KUKA KRL program: MyProgram_258().src

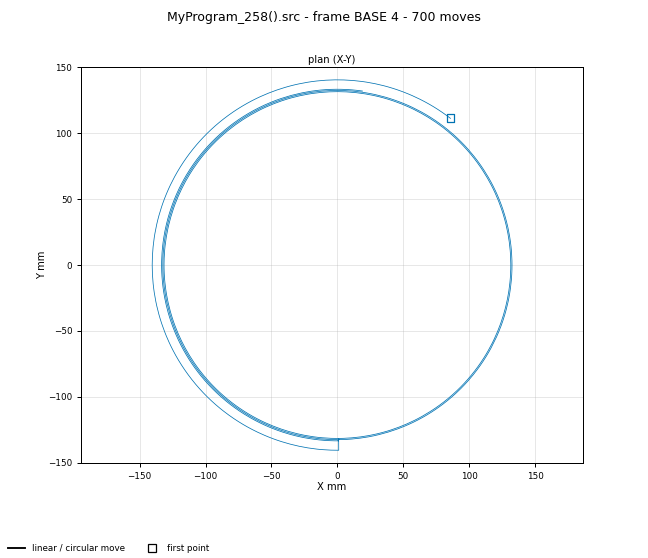
[picture p0: tool path of MyProgram_258().src in frame BASE 4, 700 of 700 moves have a stored position in this frame; points joined in program order, loops and branches not executed]
&ACCESS RVP
&REL 1
&PARAM TEMPLATE = C:\KRC\Roboter\Template\vorgabe
&PARAM EDITMASK = *
DEF MyProgram_258()
; ---- Setting reference (Base) ----
$BASE = BASE_DATA[4]

; --------------------------
; ---- Setting tool (TCP) ----
$TOOL = TOOL_DATA[3]
; --------------------------

$VEL.CP = VEL_APROX_PRINT
Startdeposition()
$VEL.CP = VEL_PRINT
LIN {X 85.7174,Y 111.2402,Z 166,A 52.9681,B 10.7255,C 0.0747,E1 10.8235,E2 398.079} C_DIS
LIN {X 83.0634,Y 113.235,Z 166,A 54.4984,B 10.7255,C 0.0678,E1 10.82,E2 396.526} C_DIS
LIN {X 79.5534,Y 115.7279,Z 166,A 56.2475,B 10.7255,C 0.0651,E1 10.816,E2 394.7774} C_DIS
LIN {X 75.9568,Y 118.12,Z 166,A 57.9765,B 10.7255,C 0.0632,E1 10.812,E2 393.0524} C_DIS
LIN {X 72.9306,Y 120.0121,Z 166,A 59.3925,B 10.7255,C 0.0621,E1 10.8086,E2 391.6413} C_DIS
LIN {X 69.966,Y 121.7647,Z 166,A 60.8768,B 10.7255,C 0.0581,E1 10.805,E2 390.1468} C_DIS
LIN {X 66.2006,Y 123.8518,Z 166,A 62.5606,B 10.7255,C 0.0575,E1 10.8009,E2 388.4721} C_DIS
LIN {X 62.4847,Y 125.7655,Z 166,A 64.2605,B 10.7256,C 0.0555,E1 10.7967,E2 386.7727} C_DIS
LIN {X 59.1907,Y 127.3486,Z 166,A 65.6969,B 10.7256,C 0.055,E1 10.7931,E2 385.3432} C_DIS
LIN {X 56.6753,Y 128.4896,Z 166,A 66.832,B 10.7256,C 0.0535,E1 10.7902,E2 384.2072} C_DIS
LIN {X 53.7331,Y 129.7462,Z 166,A 68.1368,B 10.7256,C 0.0521,E1 10.7868,E2 382.9025} C_DIS
LIN {X 49.8023,Y 131.3058,Z 166,A 69.9999,B 10.7256,C 0.0469,E1 10.7819,E2 381.0219} C_DIS
LIN {X 45.6873,Y 132.7929,Z 166,A 71.6306,B 10.7256,C 0.0491,E1 10.7777,E2 379.4111} C_DIS
LIN {X 42.4057,Y 133.877,Z 166,A 73.0559,B 10.7256,C 0.0475,E1 10.7739,E2 377.9841} C_DIS
LIN {X 38.7409,Y 134.9848,Z 166,A 74.5834,B 10.7256,C 0.0472,E1 10.7698,E2 376.4612} C_DIS
LIN {X 35.4064,Y 135.8978,Z 166,A 76.0506,B 10.7256,C 0.0448,E1 10.7658,E2 374.9871} C_DIS
LIN {X 31.4821,Y 136.8581,Z 166,A 77.4069,B 10.7256,C 0.0508,E1 10.7622,E2 373.6681} C_DIS
LIN {X 28.7539,Y 137.4591,Z 166,A 78.7425,B 10.7256,C 0.0454,E1 10.7585,E2 372.308} C_DIS
LIN {X 25.6831,Y 138.0655,Z 166,A 80.0395,B 10.7256,C 0.0443,E1 10.755,E2 371.0088} C_DIS
LIN {X 22.2954,Y 138.6535,Z 166,A 81.461,B 10.7256,C 0.0432,E1 10.751,E2 369.5854} C_DIS
LIN {X 18.6465,Y 139.1895,Z 166,A 82.9581,B 10.7256,C 0.0429,E1 10.7469,E2 368.0897} C_DIS
LIN {X 14.9704,Y 139.6322,Z 166,A 84.3565,B 10.7256,C 0.0451,E1 10.7431,E2 366.7061} C_DIS
LIN {X 11.786,Y 139.937,Z 166,A 85.7616,B 10.7256,C 0.0424,E1 10.7391,E2 365.2888} C_DIS
LIN {X 8.3535,Y 140.1841,Z 166,A 87.1286,B 10.7256,C 0.0431,E1 10.7353,E2 363.927} C_DIS
LIN {X 4.9167,Y 140.3475,Z 166,A 88.5506,B 10.7256,C 0.0426,E1 10.7314,E2 362.5033} C_DIS
LIN {X 1.7237,Y 140.4233,Z 166,A 89.9324,B 10.7256,C 0.0407,E1 10.7275,E2 361.1121} C_DIS
LIN {X -1.7428,Y 140.423,Z 166,A 91.3065,B 10.7256,C 0.0418,E1 10.7237,E2 359.7437} C_DIS
LIN {X -5.4304,Y 140.3274,Z 166,A 92.7483,B 10.7256,C 0.0434,E1 10.7197,E2 358.3106} C_DIS
LIN {X -8.7826,Y 140.1576,Z 166,A 94.1374,B 10.7256,C 0.0433,E1 10.7158,E2 356.9198} C_DIS
LIN {X -12.3639,Y 139.8881,Z 166,A 95.6189,B 10.7256,C 0.0433,E1 10.7116,E2 355.437} C_DIS
LIN {X -15.5753,Y 139.5671,Z 166,A 96.9396,B 10.7256,C 0.0437,E1 10.708,E2 354.1166} C_DIS
LIN {X -19.209,Y 139.1139,Z 166,A 98.4595,B 10.7256,C 0.0437,E1 10.7038,E2 352.5943} C_DIS
LIN {X -22.5934,Y 138.6039,Z 166,A 99.8716,B 10.7256,C 0.0441,E1 10.6999,E2 351.1811} C_DIS
LIN {X -26.0391,Y 137.9974,Z 166,A 101.2635,B 10.7256,C 0.0457,E1 10.6961,E2 349.7946} C_DIS
LIN {X -29.3329,Y 137.3349,Z 166,A 102.6588,B 10.7256,C 0.046,E1 10.6922,E2 348.397} C_DIS
LIN {X -32.6927,Y 136.5739,Z 166,A 104.0676,B 10.7256,C 0.0469,E1 10.6884,E2 346.9887} C_DIS
LIN {X -36.0321,Y 135.731,Z 166,A 105.4187,B 10.7256,C 0.0493,E1 10.6848,E2 345.6455} C_DIS
LIN {X -39.5794,Y 134.7392,Z 166,A 106.9465,B 10.7256,C 0.05,E1 10.6807,E2 344.1156} C_DIS
LIN {X -42.9868,Y 133.6913,Z 166,A 108.3925,B 10.7256,C 0.0515,E1 10.6768,E2 342.6718} C_DIS
LIN {X -45.9258,Y 132.7102,Z 166,A 109.7162,B 10.7256,C 0.0514,E1 10.6733,E2 341.3415} C_DIS
LIN {X -49.682,Y 131.3509,Z 166,A 111.2836,B 10.7256,C 0.0545,E1 10.6692,E2 339.7834} C_DIS
LIN {X -52.371,Y 130.3013,Z 166,A 112.5376,B 10.7256,C 0.0541,E1 10.6659,E2 338.5205} C_DIS
LIN {X -55.8214,Y 128.8608,Z 166,A 113.9843,B 10.7256,C 0.0577,E1 10.6623,E2 337.0851} C_DIS
LIN {X -58.4834,Y 127.6757,Z 166,A 115.2991,B 10.7256,C 0.0564,E1 10.6589,E2 335.7554} C_DIS
LIN {X -61.664,Y 126.1703,Z 166,A 116.7076,B 10.7256,C 0.0589,E1 10.6553,E2 334.3516} C_DIS
LIN {X -64.8452,Y 124.5651,Z 166,A 118.1373,B 10.7256,C 0.0614,E1 10.6518,E2 332.9262} C_DIS
LIN {X -68.498,Y 122.5963,Z 166,A 119.9049,B 10.7256,C 0.0623,E1 10.6474,E2 331.1507} C_DIS
LIN {X -72.1926,Y 120.4576,Z 166,A 121.6574,B 10.7256,C 0.0647,E1 10.6432,E2 329.3985} C_DIS
LIN {X -75.871,Y 118.1749,Z 166,A 123.4185,B 10.7256,C 0.0676,E1 10.6391,E2 327.6397} C_DIS
LIN {X -78.8459,Y 116.2112,Z 166,A 125.0176,B 10.7256,C 0.0669,E1 10.6353,E2 326.0236} C_DIS
LIN {X -82.7583,Y 113.4589,Z 166,A 126.9317,B 10.7256,C 0.0711,E1 10.631,E2 324.1162} C_DIS
LIN {X -86.3102,Y 110.7807,Z 166,A 128.7237,B 10.7255,C 0.0749,E1 10.627,E2 322.3288} C_DIS
LIN {X -89.1917,Y 108.4744,Z 166,A 130.3265,B 10.7255,C 0.0757,E1 10.6235,E2 320.7152} C_DIS
LIN {X -92.4731,Y 105.6904,Z 166,A 132.0844,B 10.7255,C 0.0791,E1 10.6198,E2 318.9588} C_DIS
LIN {X -95.6725,Y 102.803,Z 166,A 133.7492,B 10.7255,C 0.0846,E1 10.6164,E2 317.3077} C_DIS
LIN {X -98.6977,Y 99.903,Z 166,A 135.4739,B 10.7254,C 0.0879,E1 10.613,E2 315.5829} C_DIS
LIN {X -101.6253,Y 96.9226,Z 166,A 137.2193,B 10.7254,C 0.0907,E1 10.6096,E2 313.8341} C_DIS
LIN {X -104.1361,Y 94.2199,Z 166,A 138.7083,B 10.7254,C 0.0943,E1 10.6068,E2 312.3488} C_DIS
LIN {X -106.8373,Y 91.1457,Z 166,A 140.4303,B 10.7254,C 0.097,E1 10.6036,E2 310.6219} C_DIS
LIN {X -109.1132,Y 88.4087,Z 166,A 142.0079,B 10.7254,C 0.0976,E1 10.6008,E2 309.03} C_DIS
LIN {X -112.0478,Y 84.6581,Z 166,A 143.9057,B 10.7253,C 0.1032,E1 10.5976,E2 307.14} C_DIS
LIN {X -114.3919,Y 81.4632,Z 166,A 145.5929,B 10.7253,C 0.1056,E1 10.5948,E2 305.4456} C_DIS
LIN {X -116.8357,Y 77.9173,Z 166,A 147.3595,B 10.7252,C 0.1097,E1 10.592,E2 303.6797} C_DIS
LIN {X -119.1097,Y 74.3951,Z 166,A 149.0835,B 10.7252,C 0.1137,E1 10.5895,E2 301.9559} C_DIS
LIN {X -121.334,Y 70.71,Z 166,A 150.7899,B 10.7251,C 0.1193,E1 10.587,E2 300.2578} C_DIS
LIN {X -123.4441,Y 66.9578,Z 166,A 152.6788,B 10.7251,C 0.121,E1 10.5845,E2 298.354} C_DIS
LIN {X -125.2195,Y 63.5706,Z 166,A 154.115,B 10.725,C 0.1277,E1 10.5827,E2 296.9353} C_DIS
LIN {X -126.6897,Y 60.5875,Z 166,A 155.2897,B 10.725,C 0.1351,E1 10.5813,E2 295.7852} C_DIS
LIN {X -128.075,Y 57.6021,Z 166,A 156.8232,B 10.725,C 0.1348,E1 10.5795,E2 294.229} C_DIS
LIN {X -129.665,Y 53.9275,Z 166,A 158.5396,B 10.7249,C 0.1375,E1 10.5776,E2 292.5039} C_DIS
LIN {X -131.0262,Y 50.5316,Z 166,A 160.0242,B 10.7249,C 0.1418,E1 10.576,E2 291.022} C_DIS
LIN {X -132.2233,Y 47.3105,Z 166,A 161.4457,B 10.7248,C 0.1453,E1 10.5747,E2 289.5996} C_DIS
LIN {X -133.3465,Y 44.0455,Z 166,A 162.8717,B 10.7248,C 0.1489,E1 10.5734,E2 288.173} C_DIS
LIN {X -134.4583,Y 40.5278,Z 166,A 164.4487,B 10.7247,C 0.1516,E1 10.5721,E2 286.5885} C_DIS
LIN {X -135.3443,Y 37.4599,Z 166,A 165.7163,B 10.7247,C 0.1561,E1 10.5712,E2 285.3268} C_DIS
LIN {X -136.2255,Y 34.1176,Z 166,A 167.1446,B 10.7246,C 0.1597,E1 10.5702,E2 283.8977} C_DIS
LIN {X -137.0215,Y 30.7667,Z 166,A 168.5675,B 10.7246,C 0.1634,E1 10.5693,E2 282.4742} C_DIS
LIN {X -137.7352,Y 27.397,Z 166,A 169.9898,B 10.7245,C 0.1671,E1 10.5685,E2 281.0512} C_DIS
LIN {X -138.3664,Y 24.0105,Z 166,A 171.4122,B 10.7245,C 0.1708,E1 10.5678,E2 279.6282} C_DIS
LIN {X -138.9138,Y 20.6098,Z 166,A 172.9305,B 10.7244,C 0.1726,E1 10.5671,E2 278.097} C_DIS
LIN {X -139.407,Y 16.9421,Z 166,A 174.34,B 10.7243,C 0.1791,E1 10.5666,E2 276.7019} C_DIS
LIN {X -139.7635,Y 13.6928,Z 166,A 175.7816,B 10.7243,C 0.1807,E1 10.5662,E2 275.2479} C_DIS
LIN {X -140.0738,Y 10.0321,Z 166,A 177.2439,B 10.7242,C 0.1859,E1 10.5659,E2 273.7919} C_DIS
LIN {X -140.2655,Y 6.8493,Z 166,A 178.5857,B 10.7242,C 0.1888,E1 10.5657,E2 272.4462} C_DIS
LIN {X -140.4085,Y 2.6106,Z 166,A -179.8067,B 10.724,C 0.1965,E1 10.5656,E2 270.8561} C_DIS
LIN {X -140.4365,Y -0.0242,Z 166,A -178.4973,B 10.724,C 0.1948,E1 10.5656,E2 269.5179} C_DIS
LIN {X -140.3907,Y -3.4567,Z 166,A -177.1039,B 10.724,C 0.199,E1 10.5656,E2 268.1267} C_DIS
LIN {X -140.266,Y -6.8381,Z 166,A -175.7478,B 10.7238,C 0.2035,E1 10.5658,E2 266.7751} C_DIS
LIN {X -139.9886,Y -11.1743,Z 166,A -174.043,B 10.7238,C 0.2101,E1 10.5661,E2 265.0808} C_DIS
LIN {X -139.7327,Y -14.0133,Z 166,A -172.8116,B 10.7237,C 0.2121,E1 10.5665,E2 263.8418} C_DIS
LIN {X -139.3773,Y -17.1908,Z 166,A -171.436,B 10.7237,C 0.2144,E1 10.5669,E2 262.4583} C_DIS
LIN {X -138.8773,Y -20.8502,Z 166,A -169.9239,B 10.7235,C 0.2186,E1 10.5675,E2 260.947} C_DIS
LIN {X -138.2783,Y -24.503,Z 166,A -168.4632,B 10.7235,C 0.224,E1 10.5682,E2 259.494} C_DIS
LIN {X -137.685,Y -27.6437,Z 166,A -167.077,B 10.7234,C 0.226,E1 10.5689,E2 258.0985} C_DIS
LIN {X -136.9287,Y -31.1727,Z 166,A -165.623,B 10.7234,C 0.2306,E1 10.5698,E2 256.6481} C_DIS
LIN {X -136.0361,Y -34.8636,Z 166,A -164.0961,B 10.7232,C 0.2354,E1 10.5708,E2 255.1255} C_DIS
LIN {X -135.342,Y -37.4682,Z 166,A -162.9018,B 10.7232,C 0.2365,E1 10.5717,E2 253.9199} C_DIS
LIN {X -134.3111,Y -41.0087,Z 166,A -161.3782,B 10.7231,C 0.2403,E1 10.5729,E2 252.3951} C_DIS
LIN {X -133.2661,Y -44.2868,Z 166,A -159.9559,B 10.7231,C 0.2438,E1 10.5742,E2 250.9716} C_DIS
LIN {X -132.1411,Y -47.5382,Z 166,A -158.534,B 10.7229,C 0.2472,E1 10.5755,E2 249.5485} C_DIS
LIN {X -130.9367,Y -50.7616,Z 166,A -157.0359,B 10.7229,C 0.249,E1 10.577,E2 248.0393} C_DIS
LIN {X -129.6473,Y -53.9697,Z 166,A -155.5789,B 10.7229,C 0.2518,E1 10.5786,E2 246.5775} C_DIS
LIN {X -127.7265,Y -58.3735,Z 166,A -153.6315,B 10.7227,C 0.2573,E1 10.5808,E2 244.6333} C_DIS
LIN {X -126.2024,Y -61.599,Z 166,A -152.2299,B 10.7226,C 0.2622,E1 10.5825,E2 243.2396} C_DIS
LIN {X -124.5972,Y -64.7841,Z 166,A -150.7803,B 10.7225,C 0.2661,E1 10.5843,E2 241.7917} C_DIS
LIN {X -122.6149,Y -68.4648,Z 166,A -148.9967,B 10.7225,C 0.2687,E1 10.5867,E2 239.9993} C_DIS
LIN {X -120.4574,Y -72.1929,Z 166,A -147.1417,B 10.7224,C 0.2709,E1 10.5893,E2 238.1328} C_DIS
LIN {X -118.111,Y -75.9708,Z 166,A -145.269,B 10.7223,C 0.2741,E1 10.5922,E2 236.2537} C_DIS
LIN {X -115.7286,Y -79.5524,Z 166,A -143.5007,B 10.7222,C 0.2779,E1 10.5949,E2 234.4846} C_DIS
LIN {X -113.2061,Y -83.1027,Z 166,A -141.7158,B 10.7221,C 0.2819,E1 10.5978,E2 232.6996} C_DIS
LIN {X -110.479,Y -86.6953,Z 166,A -139.881,B 10.722,C 0.2861,E1 10.601,E2 230.8665} C_DIS
LIN {X -107.5054,Y -90.3564,Z 166,A -137.994,B 10.7218,C 0.2912,E1 10.6043,E2 228.9854} C_DIS
LIN {X -104.6071,Y -93.6965,Z 166,A -136.1896,B 10.7218,C 0.295,E1 10.6076,E2 227.1817} C_DIS
LIN {X -101.7035,Y -96.8408,Z 166,A -134.3395,B 10.7218,C 0.2963,E1 10.6112,E2 225.3188} C_DIS
LIN {X -98.6888,Y -99.9119,Z 166,A -132.5285,B 10.7216,C 0.2986,E1 10.6148,E2 223.5014} C_DIS
LIN {X -95.5786,Y -102.8905,Z 166,A -130.851,B 10.7216,C 0.3037,E1 10.6182,E2 221.8349} C_DIS
LIN {X -92.3556,Y -105.7928,Z 166,A -129.0546,B 10.7214,C 0.3064,E1 10.6219,E2 220.0355} C_DIS
LIN {X -89.088,Y -108.5591,Z 166,A -127.3599,B 10.7214,C 0.3107,E1 10.6256,E2 218.3481} C_DIS
LIN {X -86.3015,Y -110.7874,Z 166,A -125.75,B 10.7214,C 0.3097,E1 10.6291,E2 216.7185} C_DIS
LIN {X -82.3699,Y -113.7404,Z 166,A -123.764,B 10.7212,C 0.3135,E1 10.6336,E2 214.7356} C_DIS
LIN {X -78.5505,Y -116.4111,Z 166,A -121.8547,B 10.7212,C 0.3163,E1 10.638,E2 212.8257} C_DIS
LIN {X -75.1269,Y -118.6494,Z 166,A -120.1443,B 10.7211,C 0.3178,E1 10.642,E2 211.11} C_DIS
LIN {X -71.4556,Y -120.8964,Z 166,A -118.5045,B 10.7209,C 0.3229,E1 10.6459,E2 209.4857} C_DIS
LIN {X -68.3612,Y -122.6727,Z 166,A -116.8962,B 10.7209,C 0.3214,E1 10.6499,E2 207.8575} C_DIS
LIN {X -64.569,Y -124.7101,Z 166,A -115.1164,B 10.7209,C 0.323,E1 10.6543,E2 206.0747} C_DIS
LIN {X -60.6866,Y -126.6424,Z 166,A -113.492,B 10.7208,C 0.3284,E1 10.6583,E2 204.4693} C_DIS
LIN {X -57.686,Y -128.0375,Z 166,A -112.3048,B 10.7206,C 0.3337,E1 10.6613,E2 203.3034} C_DIS
LIN {X -55.323,Y -129.0763,Z 166,A -111.0698,B 10.7207,C 0.3306,E1 10.6645,E2 202.0446} C_DIS
LIN {X -52.1431,Y -130.3932,Z 166,A -109.6601,B 10.7207,C 0.3319,E1 10.6681,E2 200.6342} C_DIS
LIN {X -48.9322,Y -131.6317,Z 166,A -108.249,B 10.7207,C 0.333,E1 10.6718,E2 199.222} C_DIS
LIN {X -45.6787,Y -132.7958,Z 166,A -106.8356,B 10.7207,C 0.3341,E1 10.6756,E2 197.8079} C_DIS
LIN {X -42.3173,Y -133.9052,Z 166,A -105.3701,B 10.7206,C 0.3347,E1 10.6795,E2 196.3394} C_DIS
LIN {X -38.8146,Y -134.9632,Z 166,A -103.9003,B 10.7206,C 0.3363,E1 10.6834,E2 194.8725} C_DIS
LIN {X -35.7228,Y -135.8135,Z 166,A -102.5809,B 10.7206,C 0.3369,E1 10.687,E2 193.5514} C_DIS
LIN {X -31.9412,Y -136.7532,Z 166,A -101.0442,B 10.7205,C 0.3391,E1 10.6911,E2 192.0213} C_DIS
LIN {X -29.0661,Y -137.3925,Z 166,A -99.784,B 10.7205,C 0.3383,E1 10.6946,E2 190.7531} C_DIS
LIN {X -25.6925,Y -138.0637,Z 166,A -98.3811,B 10.7205,C 0.3389,E1 10.6984,E2 189.3499} C_DIS
LIN {X -22.3036,Y -138.6522,Z 166,A -96.9553,B 10.7205,C 0.3389,E1 10.7024,E2 187.9208} C_DIS
LIN {X -18.6541,Y -139.1885,Z 166,A -95.4474,B 10.7205,C 0.3392,E1 10.7065,E2 186.412} C_DIS
LIN {X -15.465,Y -139.5789,Z 166,A -94.1374,B 10.7205,C 0.3395,E1 10.7102,E2 185.1016} C_DIS
LIN {X -11.7927,Y -139.9364,Z 166,A -92.6422,B 10.7205,C 0.3399,E1 10.7143,E2 183.6071} C_DIS
LIN {X -8.3593,Y -140.1837,Z 166,A -91.2738,B 10.7204,C 0.3409,E1 10.7181,E2 182.2429} C_DIS
LIN {X -4.9207,Y -140.3473,Z 166,A -89.8498,B 10.7204,C 0.3404,E1 10.7221,E2 180.8157} C_DIS
LIN {X -1.71,Y -140.4235,Z 166,A -88.4652,B 10.7204,C 0.3385,E1 10.726,E2 179.4207} C_DIS
LIN {X 0.9985,Y -140.4282,Z 166,A -87.7382,B 10.7202,C 0.3476,E1 10.7279,E2 178.7427} C_DIS
Enddeposition()
LIN {X 0.9528,Y -131.4631,Z 167,A -88.3932,B 11.3356,C 0.2691,E1 11.3404,E2 178.9455} C_DIS
Startdeposition()
$VEL.CP = VEL_PRINT
LIN {X -1.6196,Y -131.4601,Z 167,A -89.776,B 11.3354,C 0.2755,E1 11.3364,E2 180.3603} C_DIS
LIN {X -4.8405,Y -131.38,Z 167,A -91.1508,B 11.3354,C 0.2748,E1 11.3326,E2 181.7322} C_DIS
LIN {X -8.4656,Y -131.1965,Z 167,A -92.6004,B 11.3355,C 0.2717,E1 11.3286,E2 183.1667} C_DIS
LIN {X -11.6768,Y -130.9506,Z 167,A -94.0267,B 11.3355,C 0.2721,E1 11.3246,E2 184.5963} C_DIS
LIN {X -14.4963,Y -130.6678,Z 167,A -95.3539,B 11.3355,C 0.274,E1 11.3209,E2 185.935} C_DIS
LIN {X -18.0814,Y -130.2204,Z 167,A -96.8808,B 11.3355,C 0.2725,E1 11.3167,E2 187.4567} C_DIS
LIN {X -21.2806,Y -129.7354,Z 167,A -98.2888,B 11.3355,C 0.272,E1 11.3128,E2 188.8648} C_DIS
LIN {X -24.4682,Y -129.1718,Z 167,A -99.5735,B 11.3355,C 0.2685,E1 11.3093,E2 190.1348} C_DIS
LIN {X -27.6142,Y -128.5358,Z 167,A -101.1,B 11.3355,C 0.2708,E1 11.3051,E2 191.677} C_DIS
LIN {X -30.3791,Y -127.9112,Z 167,A -102.3409,B 11.3355,C 0.2702,E1 11.3017,E2 192.9189} C_DIS
LIN {X -33.8824,Y -127.0274,Z 167,A -103.9798,B 11.3355,C 0.2707,E1 11.2972,E2 194.5657} C_DIS
LIN {X -37.0063,Y -126.1527,Z 167,A -105.3341,B 11.3355,C 0.2684,E1 11.2936,E2 195.9132} C_DIS
LIN {X -39.7094,Y -125.3284,Z 167,A -106.5704,B 11.3356,C 0.2676,E1 11.2903,E2 197.1502} C_DIS
LIN {X -42.7754,Y -124.3153,Z 167,A -107.9828,B 11.3356,C 0.2666,E1 11.2866,E2 198.5634} C_DIS
LIN {X -45.8088,Y -123.2299,Z 167,A -109.392,B 11.3356,C 0.2654,E1 11.2829,E2 199.9733} C_DIS
LIN {X -48.8167,Y -122.0696,Z 167,A -110.802,B 11.3356,C 0.2642,E1 11.2792,E2 201.384} C_DIS
LIN {X -51.8039,Y -120.8323,Z 167,A -112.2163,B 11.3357,C 0.2629,E1 11.2756,E2 202.799} C_DIS
LIN {X -54.7506,Y -119.5262,Z 167,A -113.6279,B 11.3357,C 0.2615,E1 11.272,E2 204.2114} C_DIS
LIN {X -57.8494,Y -118.0571,Z 167,A -115.0803,B 11.3358,C 0.2588,E1 11.2683,E2 205.6587} C_DIS
LIN {X -60.8996,Y -116.5127,Z 167,A -116.4678,B 11.3359,C 0.2548,E1 11.2649,E2 207.0339} C_DIS
LIN {X -64.05,Y -114.8138,Z 167,A -118.31,B 11.3359,C 0.259,E1 11.2603,E2 208.9097} C_DIS
LIN {X -67.5842,Y -112.7693,Z 167,A -119.9987,B 11.3359,C 0.2545,E1 11.2563,E2 210.5874} C_DIS
LIN {X -70.671,Y -110.8608,Z 167,A -121.6957,B 11.3359,C 0.2547,E1 11.2522,E2 212.2979} C_DIS
LIN {X -74.39,Y -108.4,Z 167,A -123.6086,B 11.3359,C 0.2511,E1 11.2478,E2 214.2068} C_DIS
LIN {X -77.0224,Y -106.5458,Z 167,A -124.9509,B 11.3361,C 0.2475,E1 11.2448,E2 215.5415} C_DIS
LIN {X -80.0944,Y -104.2564,Z 167,A -126.6676,B 11.3361,C 0.2457,E1 11.2409,E2 217.2633} C_DIS
LIN {X -83.2482,Y -101.7555,Z 167,A -128.4689,B 11.3361,C 0.2437,E1 11.237,E2 219.0697} C_DIS
LIN {X -86.4707,Y -99.0316,Z 167,A -130.3006,B 11.3362,C 0.2402,E1 11.2331,E2 220.9} C_DIS
LIN {X -89.4839,Y -96.3177,Z 167,A -132.0835,B 11.3362,C 0.2371,E1 11.2295,E2 222.6842} C_DIS
LIN {X -92.3941,Y -93.5302,Z 167,A -133.9462,B 11.3363,C 0.2359,E1 11.2257,E2 224.5588} C_DIS
LIN {X -95.3517,Y -90.5132,Z 167,A -135.8075,B 11.3363,C 0.2326,E1 11.2221,E2 226.4216} C_DIS
LIN {X -98.3569,Y -87.2376,Z 167,A -137.6719,B 11.3365,C 0.227,E1 11.2186,E2 228.2766} C_DIS
LIN {X -101.2512,Y -83.8608,Z 167,A -139.6968,B 11.3365,C 0.2246,E1 11.215,E2 230.3107} C_DIS
LIN {X -104.0256,Y -80.3937,Z 167,A -141.5014,B 11.3367,C 0.2176,E1 11.2119,E2 232.0988} C_DIS
LIN {X -105.9668,Y -77.8169,Z 167,A -143.0743,B 11.3367,C 0.2178,E1 11.2092,E2 233.6906} C_DIS
LIN {X -108.6249,Y -74.0623,Z 167,A -144.9383,B 11.3368,C 0.2102,E1 11.2063,E2 235.537} C_DIS
LIN {X -110.294,Y -71.5519,Z 167,A -146.3582,B 11.3368,C 0.2092,E1 11.2041,E2 236.9685} C_DIS
LIN {X -112.1328,Y -68.6344,Z 167,A -147.8428,B 11.3368,C 0.2052,E1 11.2019,E2 238.45} C_DIS
LIN {X -113.7899,Y -65.8505,Z 167,A -149.2653,B 11.337,C 0.2019,E1 11.1999,E2 239.8728} C_DIS
LIN {X -115.3682,Y -63.0446,Z 167,A -150.5965,B 11.337,C 0.1969,E1 11.1981,E2 241.1945} C_DIS
LIN {X -116.8769,Y -60.2004,Z 167,A -152.146,B 11.337,C 0.1963,E1 11.196,E2 242.7602} C_DIS
LIN {X -118.1647,Y -57.6313,Z 167,A -153.4289,B 11.337,C 0.1937,E1 11.1945,E2 244.0459} C_DIS
LIN {X -119.7507,Y -54.2596,Z 167,A -154.9749,B 11.3372,C 0.1878,E1 11.1927,E2 245.5815} C_DIS
LIN {X -120.9894,Y -51.4404,Z 167,A -156.3794,B 11.3372,C 0.1856,E1 11.1911,E2 246.9923} C_DIS
LIN {X -122.2209,Y -48.4413,Z 167,A -157.8015,B 11.3372,C 0.1819,E1 11.1896,E2 248.4144} C_DIS
LIN {X -123.3708,Y -45.4326,Z 167,A -159.2278,B 11.3373,C 0.1786,E1 11.1882,E2 249.8422} C_DIS
LIN {X -124.4468,Y -42.3962,Z 167,A -160.6477,B 11.3373,C 0.1751,E1 11.1869,E2 251.2629} C_DIS
LIN {X -125.649,Y -38.6824,Z 167,A -162.5181,B 11.3374,C 0.1737,E1 11.1853,E2 253.1516} C_DIS
LIN {X -126.7149,Y -35.0351,Z 167,A -164.0453,B 11.3375,C 0.1665,E1 11.1842,E2 254.6622} C_DIS
LIN {X -127.6297,Y -31.5469,Z 167,A -165.7364,B 11.3375,C 0.1645,E1 11.183,E2 256.3659} C_DIS
LIN {X -128.3549,Y -28.4521,Z 167,A -167.0588,B 11.3376,C 0.1593,E1 11.1822,E2 257.6797} C_DIS
LIN {X -128.9411,Y -25.6615,Z 167,A -168.2945,B 11.3376,C 0.1556,E1 11.1815,E2 258.9134} C_DIS
LIN {X -129.5291,Y -22.5087,Z 167,A -169.7075,B 11.3377,C 0.1519,E1 11.1808,E2 260.3269} C_DIS
LIN {X -130.0472,Y -19.2933,Z 167,A -171.1719,B 11.3377,C 0.1487,E1 11.1801,E2 261.7952} C_DIS
LIN {X -130.5424,Y -15.5789,Z 167,A -172.7879,B 11.3378,C 0.1436,E1 11.1796,E2 263.4075} C_DIS
LIN {X -130.8365,Y -12.8823,Z 167,A -174.0944,B 11.3378,C 0.1426,E1 11.1792,E2 264.7274} C_DIS
LIN {X -131.1127,Y -9.6697,Z 167,A -175.4356,B 11.3379,C 0.1372,E1 11.1789,E2 266.0597} C_DIS
LIN {X -131.33,Y -6.063,Z 167,A -176.9873,B 11.3379,C 0.1321,E1 11.1787,E2 267.6072} C_DIS
LIN {X -131.4446,Y -2.5537,Z 167,A -178.6248,B 11.3379,C 0.1298,E1 11.1785,E2 269.2556} C_DIS
LIN {X -131.4667,Y 0.7845,Z 167,A 179.8914,B 11.338,C 0.1261,E1 11.1785,E2 270.7413} C_DIS
LIN {X -131.3681,Y 5.147,Z 167,A 178.0051,B 11.338,C 0.1202,E1 11.1787,E2 272.6237} C_DIS
LIN {X -131.1977,Y 8.4457,Z 167,A 176.6123,B 11.3382,C 0.115,E1 11.1789,E2 274.0096} C_DIS
LIN {X -130.9508,Y 11.6749,Z 167,A 175.1443,B 11.3382,C 0.112,E1 11.1793,E2 275.4827} C_DIS
LIN {X -130.6588,Y 14.5795,Z 167,A 173.7611,B 11.3382,C 0.1105,E1 11.1797,E2 276.8774} C_DIS
LIN {X -130.2126,Y 18.1359,Z 167,A 172.2485,B 11.3382,C 0.1049,E1 11.1802,E2 278.3825} C_DIS
LIN {X -129.7327,Y 21.297,Z 167,A 170.8374,B 11.3382,C 0.1012,E1 11.1808,E2 279.7941} C_DIS
LIN {X -129.1745,Y 24.4542,Z 167,A 169.5469,B 11.3383,C 0.095,E1 11.1815,E2 281.0707} C_DIS
LIN {X -128.528,Y 27.6503,Z 167,A 167.9884,B 11.3383,C 0.0936,E1 11.1824,E2 282.6436} C_DIS
LIN {X -127.909,Y 30.3884,Z 167,A 166.7412,B 11.3383,C 0.0906,E1 11.1831,E2 283.8921} C_DIS
LIN {X -127.0251,Y 33.8909,Z 167,A 165.2467,B 11.3384,C 0.0845,E1 11.1842,E2 285.3755} C_DIS
LIN {X -126.2662,Y 36.6186,Z 167,A 163.8979,B 11.3384,C 0.0832,E1 11.1852,E2 286.7364} C_DIS
LIN {X -125.3302,Y 39.7039,Z 167,A 162.4751,B 11.3384,C 0.0796,E1 11.1864,E2 288.1596} C_DIS
LIN {X -124.3192,Y 42.7642,Z 167,A 161.053,B 11.3384,C 0.076,E1 11.1877,E2 289.5822} C_DIS
LIN {X -123.2341,Y 45.7975,Z 167,A 159.629,B 11.3384,C 0.0725,E1 11.189,E2 291.0068} C_DIS
LIN {X -122.0036,Y 48.9805,Z 167,A 158.1656,B 11.3385,C 0.0679,E1 11.1905,E2 292.4658} C_DIS
LIN {X -120.8275,Y 51.8149,Z 167,A 156.7749,B 11.3385,C 0.0653,E1 11.192,E2 293.8612} C_DIS
LIN {X -119.5263,Y 54.7504,Z 167,A 155.3549,B 11.3385,C 0.0619,E1 11.1936,E2 295.282} C_DIS
LIN {X -118.1452,Y 57.6709,Z 167,A 153.9342,B 11.3385,C 0.0584,E1 11.1954,E2 296.7026} C_DIS
LIN {X -116.4688,Y 60.9832,Z 167,A 152.4919,B 11.3386,C 0.0506,E1 11.1972,E2 298.1226} C_DIS
LIN {X -115.1796,Y 63.3893,Z 167,A 151.092,B 11.3386,C 0.0517,E1 11.1991,E2 299.5456} C_DIS
LIN {X -113.5928,Y 66.1911,Z 167,A 149.6609,B 11.3386,C 0.0486,E1 11.2011,E2 300.9783} C_DIS
LIN {X -111.9361,Y 68.9551,Z 167,A 148.1718,B 11.3386,C 0.0468,E1 11.2032,E2 302.4757} C_DIS
LIN {X -109.5762,Y 72.6476,Z 167,A 146.2018,B 11.3386,C 0.0432,E1 11.2062,E2 304.4505} C_DIS
LIN {X -107.2584,Y 76.0275,Z 167,A 144.574,B 11.3386,C 0.0356,E1 11.2088,E2 306.0579} C_DIS
LIN {X -105.5966,Y 78.3189,Z 167,A 143.1404,B 11.3386,C 0.0367,E1 11.2112,E2 307.5133} C_DIS
LIN {X -103.1467,Y 81.5191,Z 167,A 141.3473,B 11.3386,C 0.0333,E1 11.2143,E2 309.3087} C_DIS
LIN {X -100.4654,Y 84.8014,Z 167,A 139.4835,B 11.3386,C 0.0294,E1 11.2176,E2 311.1724} C_DIS
LIN {X -97.8204,Y 87.8386,Z 167,A 137.7229,B 11.3386,C 0.0255,E1 11.2209,E2 312.9317} C_DIS
LIN {X -95.0841,Y 90.7935,Z 167,A 135.9585,B 11.3387,C 0.0219,E1 11.2242,E2 314.6952} C_DIS
LIN {X -91.9484,Y 93.9678,Z 167,A 134.0438,B 11.3387,C 0.0172,E1 11.228,E2 316.6045} C_DIS
LIN {X -88.8833,Y 96.8721,Z 167,A 132.1318,B 11.3387,C 0.0149,E1 11.2319,E2 318.5229} C_DIS
LIN {X -85.8738,Y 99.5497,Z 167,A 130.3725,B 11.3387,C 0.0115,E1 11.2356,E2 320.2807} C_DIS
LIN {X -82.7725,Y 102.1433,Z 167,A 128.5482,B 11.3387,C 0.0094,E1 11.2396,E2 322.1104} C_DIS
LIN {X -79.2916,Y 104.868,Z 167,A 126.7615,B 11.3387,C 0.0029,E1 11.2435,E2 323.8791} C_DIS
LIN {X -77.0136,Y 106.5522,Z 167,A 125.4468,B 11.3387,C 0.0024,E1 11.2465,E2 325.2018} C_DIS
LIN {X -74.0585,Y 108.6275,Z 167,A 123.9775,B 11.3387,C -0.0025,E1 11.2498,E2 326.6575} C_DIS
LIN {X -71.69,Y 110.2043,Z 167,A 122.6027,B 11.3387,C -0.0017,E1 11.253,E2 328.0467} C_DIS
LIN {X -68.53,Y 112.1969,Z 167,A 121.038,B 11.3387,C -0.0057,E1 11.2567,E2 329.6025} C_DIS
LIN {X -65.8044,Y 113.8166,Z 167,A 119.6477,B 11.3387,C -0.0076,E1 11.2601,E2 330.9925} C_DIS
LIN {X -62.7673,Y 115.5195,Z 167,A 118.2627,B 11.3387,C -0.0127,E1 11.2634,E2 332.3608} C_DIS
LIN {X -60.1896,Y 116.8824,Z 167,A 116.8488,B 11.3387,C -0.0114,E1 11.267,E2 333.7901} C_DIS
LIN {X -57.6673,Y 118.147,Z 167,A 115.5558,B 11.3387,C -0.0117,E1 11.2702,E2 335.0894} C_DIS
LIN {X -54.3786,Y 119.6974,Z 167,A 114.0139,B 11.3387,C -0.0147,E1 11.2741,E2 336.625} C_DIS
LIN {X -51.4313,Y 120.9934,Z 167,A 112.5912,B 11.3387,C -0.016,E1 11.2778,E2 338.0488} C_DIS
LIN {X -48.4525,Y 122.2164,Z 167,A 111.1902,B 11.3387,C -0.0176,E1 11.2814,E2 339.4484} C_DIS
LIN {X -45.4293,Y 123.372,Z 167,A 109.7663,B 11.3387,C -0.0189,E1 11.2851,E2 340.8727} C_DIS
LIN {X -42.3564,Y 124.4606,Z 167,A 108.3407,B 11.3387,C -0.0202,E1 11.2889,E2 342.2977} C_DIS
LIN {X -38.5188,Y 125.6991,Z 167,A 106.5767,B 11.3387,C -0.0217,E1 11.2936,E2 344.0612} C_DIS
LIN {X -35.0609,Y 126.7077,Z 167,A 105.0021,B 11.3387,C -0.023,E1 11.2978,E2 345.6352} C_DIS
LIN {X -31.5772,Y 127.6224,Z 167,A 103.4314,B 11.3387,C -0.0242,E1 11.302,E2 347.2049} C_DIS
LIN {X -28.8204,Y 128.2715,Z 167,A 102.1237,B 11.3387,C -0.0234,E1 11.3056,E2 348.5203} C_DIS
LIN {X -25.6459,Y 128.9442,Z 167,A 100.7757,B 11.3387,C -0.0258,E1 11.3093,E2 349.8597} C_DIS
LIN {X -22.4753,Y 129.5351,Z 167,A 99.3678,B 11.3387,C -0.0266,E1 11.3131,E2 351.2669} C_DIS
LIN {X -19.2808,Y 130.049,Z 167,A 97.9318,B 11.3387,C -0.0266,E1 11.3171,E2 352.7051} C_DIS
LIN {X -15.6987,Y 130.5281,Z 167,A 96.3658,B 11.3387,C -0.0276,E1 11.3214,E2 354.269} C_DIS
LIN {X -12.8824,Y 130.8365,Z 167,A 95.0472,B 11.3387,C -0.0261,E1 11.3251,E2 355.5966} C_DIS
LIN {X -9.2633,Y 131.1424,Z 167,A 93.608,B 11.3387,C -0.0298,E1 11.3291,E2 357.0184} C_DIS
LIN {X -6.0472,Y 131.3308,Z 167,A 92.1619,B 11.3387,C -0.0291,E1 11.3331,E2 358.4687} C_DIS
LIN {X -2.8271,Y 131.44,Z 167,A 90.7992,B 11.3387,C -0.0303,E1 11.3369,E2 359.8259} C_DIS
LIN {X 0.3912,Y 131.4687,Z 167,A 89.4405,B 11.3387,C -0.0314,E1 11.3407,E2 361.1788} C_DIS
LIN {X 3.6152,Y 131.4192,Z 167,A 88.0108,B 11.3387,C -0.0308,E1 11.3447,E2 362.6107} C_DIS
LIN {X 6.8517,Y 131.2904,Z 167,A 86.4628,B 11.3387,C -0.0276,E1 11.3491,E2 364.174} C_DIS
LIN {X 11.6749,Y 130.9508,Z 167,A 84.4421,B 11.3387,C -0.0292,E1 11.3547,E2 366.1838} C_DIS
LIN {X 14.4913,Y 130.6683,Z 167,A 83.1183,B 11.3387,C -0.0268,E1 11.3584,E2 367.5177} C_DIS
LIN {X 18.3984,Y 130.1751,Z 167,A 81.547,B 11.3387,C -0.0296,E1 11.3627,E2 369.0716} C_DIS
LIN {X 21.2776,Y 129.7359,Z 167,A 80.1914,B 11.3387,C -0.027,E1 11.3664,E2 370.4368} C_DIS
LIN {X 24.4518,Y 129.1749,Z 167,A 78.914,B 11.3387,C -0.0294,E1 11.3699,E2 371.699} C_DIS
LIN {X 27.6117,Y 128.5364,Z 167,A 77.3922,B 11.3387,C -0.0259,E1 11.3741,E2 373.2341} C_DIS
LIN {X 31.2848,Y 127.6929,Z 167,A 75.6104,B 11.3387,C -0.0215,E1 11.379,E2 375.0318} C_DIS
LIN {X 35.0741,Y 126.704,Z 167,A 74.0532,B 11.3387,C -0.0239,E1 11.3831,E2 376.5713} C_DIS
LIN {X 38.6885,Y 125.6471,Z 167,A 72.3213,B 11.3387,C -0.0204,E1 11.3878,E2 378.3135} C_DIS
LIN {X 42.772,Y 124.3165,Z 167,A 70.5547,B 11.3387,C -0.0213,E1 11.3924,E2 380.0677} C_DIS
LIN {X 45.8054,Y 123.2311,Z 167,A 69.1574,B 11.3387,C -0.0201,E1 11.3961,E2 381.4641} C_DIS
LIN {X 48.8231,Y 122.067,Z 167,A 67.7548,B 11.3387,C -0.0188,E1 11.3998,E2 382.8657} C_DIS
LIN {X 51.8012,Y 120.8335,Z 167,A 66.3581,B 11.3387,C -0.0175,E1 11.4033,E2 384.2615} C_DIS
LIN {X 54.7503,Y 119.5263,Z 167,A 64.9617,B 11.3387,C -0.0161,E1 11.4069,E2 385.6568} C_DIS
LIN {X 57.6741,Y 118.1436,Z 167,A 63.5616,B 11.3387,C -0.0146,E1 11.4104,E2 387.0558} C_DIS
LIN {X 60.8948,Y 116.5152,Z 167,A 62.1545,B 11.3387,C -0.0166,E1 11.4139,E2 388.4437} C_DIS
LIN {X 63.3906,Y 115.179,Z 167,A 60.6617,B 11.3387,C -0.0086,E1 11.4176,E2 389.9669} C_DIS
LIN {X 66.2056,Y 113.5844,Z 167,A 59.3587,B 11.3387,C -0.0092,E1 11.4207,E2 391.2576} C_DIS
LIN {X 68.9706,Y 111.9266,Z 167,A 57.8847,B 11.3387,C -0.0054,E1 11.4243,E2 392.7398} C_DIS
LIN {X 72.0442,Y 109.9734,Z 167,A 56.4564,B 11.3387,C -0.0069,E1 11.4276,E2 394.1499} C_DIS
LIN {X 74.3878,Y 108.4015,Z 167,A 55.1058,B 11.3387,C -0.0019,E1 11.4307,E2 395.5148} C_DIS
LIN {X 77.0187,Y 106.5485,Z 167,A 53.7845,B 11.3387,C -0.0016,E1 11.4337,E2 396.827} C_DIS
LIN {X 80.0882,Y 104.2611,Z 167,A 52.0951,B 11.3387,C 0.0018,E1 11.4375,E2 398.5193} C_DIS
LIN {X 83.2529,Y 101.7516,Z 167,A 50.3166,B 11.3387,C 0.0054,E1 11.4414,E2 400.3005} C_DIS
LIN {X 86.4896,Y 99.0151,Z 167,A 48.5121,B 11.3387,C 0.0078,E1 11.4452,E2 402.1006} C_DIS
LIN {X 89.4826,Y 96.3188,Z 167,A 46.7664,B 11.3387,C 0.0109,E1 11.4488,E2 403.8457} C_DIS
LIN {X 92.3923,Y 93.532,Z 167,A 44.9375,B 11.3387,C 0.0163,E1 11.4525,E2 405.6839} C_DIS
LIN {X 95.3484,Y 90.5168,Z 167,A 43.1112,B 11.3387,C 0.0198,E1 11.456,E2 407.5093} C_DIS
LIN {X 98.361,Y 87.233,Z 167,A 41.2775,B 11.3387,C 0.0212,E1 11.4594,E2 409.3312} C_DIS
LIN {X 101.01,Y 84.152,Z 167,A 39.4485,B 11.3387,C 0.0266,E1 11.4627,E2 411.1679} C_DIS
LIN {X 103.6514,Y 80.8764,Z 167,A 37.6608,B 11.3387,C 0.0295,E1 11.4658,E2 412.9512} C_DIS
LIN {X 105.8275,Y 78.0066,Z 167,A 36.0815,B 11.3387,C 0.0334,E1 11.4685,E2 414.5325} C_DIS
LIN {X 108.4111,Y 74.3738,Z 167,A 34.2763,B 11.3387,C 0.0345,E1 11.4713,E2 416.3227} C_DIS
LIN {X 110.2022,Y 71.6933,Z 167,A 32.8055,B 11.3387,C 0.0396,E1 11.4736,E2 417.802} C_DIS
LIN {X 112.1523,Y 68.6028,Z 167,A 31.3104,B 11.3387,C 0.041,E1 11.4758,E2 419.2867} C_DIS
LIN {X 113.7929,Y 65.8454,Z 167,A 29.9299,B 11.3387,C 0.0441,E1 11.4777,E2 420.666} C_DIS
LIN {X 115.3675,Y 63.046,Z 167,A 28.6315,B 11.3387,C 0.045,E1 11.4795,E2 421.9535} C_DIS
LIN {X 116.8732,Y 60.2077,Z 167,A 27.1488,B 11.3387,C 0.0507,E1 11.4814,E2 423.4468} C_DIS
LIN {X 118.1505,Y 57.66,Z 167,A 25.8675,B 11.3386,C 0.055,E1 11.483,E2 424.7337} C_DIS
LIN {X 119.6905,Y 54.3941,Z 167,A 24.3833,B 11.3386,C 0.0568,E1 11.4847,E2 426.2086} C_DIS
LIN {X 121.0003,Y 51.4152,Z 167,A 22.9743,B 11.3386,C 0.0604,E1 11.4863,E2 427.6176} C_DIS
LIN {X 122.2212,Y 48.4407,Z 167,A 21.388,B 11.3386,C 0.069,E1 11.488,E2 429.2268} C_DIS
LIN {X 123.3697,Y 45.4356,Z 167,A 20.2064,B 11.3386,C 0.0671,E1 11.4891,E2 430.3836} C_DIS
LIN {X 124.4447,Y 42.4024,Z 167,A 18.8216,B 11.3386,C 0.0705,E1 11.4904,E2 431.7675} C_DIS
LIN {X 125.6982,Y 38.5217,Z 167,A 16.9638,B 11.3385,C 0.0775,E1 11.492,E2 433.6363} C_DIS
LIN {X 126.9375,Y 34.2192,Z 167,A 15.0026,B 11.3385,C 0.0833,E1 11.4934,E2 435.6003} C_DIS
LIN {X 127.9134,Y 30.3702,Z 167,A 13.4369,B 11.3385,C 0.0839,E1 11.4945,E2 437.1481} C_DIS
LIN {X 128.7008,Y 26.842,Z 167,A 11.9407,B 11.3385,C 0.0863,E1 11.4953,E2 438.6364} C_DIS
LIN {X 129.2491,Y 24.064,Z 167,A 10.6692,B 11.3384,C 0.0908,E1 11.496,E2 439.9136} C_DIS
LIN {X 129.8013,Y 20.8859,Z 167,A 9.2093,B 11.3384,C 0.0963,E1 11.4967,E2 441.3812} C_DIS
LIN {X 130.2753,Y 17.6841,Z 167,A 7.7714,B 11.3383,C 0.1011,E1 11.4973,E2 442.8237} C_DIS
LIN {X 130.7106,Y 14.0984,Z 167,A 6.4177,B 11.3383,C 0.0999,E1 11.4977,E2 444.1528} C_DIS
LIN {X 131.0171,Y 10.8902,Z 167,A 5.0112,B 11.3383,C 0.1041,E1 11.498,E2 445.5609} C_DIS
LIN {X 131.2212,Y 8.0646,Z 167,A 3.6729,B 11.3382,C 0.1104,E1 11.4983,E2 446.9127} C_DIS
LIN {X 131.4163,Y 3.718,Z 167,A 2.0773,B 11.3382,C 0.108,E1 11.4985,E2 448.4746} C_DIS
LIN {X 131.467,Y 0.7331,Z 167,A 0.5845,B 11.3382,C 0.117,E1 11.4985,E2 449.9915} C_DIS
LIN {X 131.4399,Y -2.8368,Z 167,A -1.0783,B 11.3381,C 0.1244,E1 11.4985,E2 451.6687} C_DIS
LIN {X 131.2913,Y -6.8338,Z 167,A -2.6834,B 11.3381,C 0.1259,E1 11.4983,E2 453.2593} C_DIS
LIN {X 131.1121,Y -9.6781,Z 167,A -3.9561,B 11.338,C 0.1303,E1 11.498,E2 454.537} C_DIS
LIN {X 130.7962,Y -13.3015,Z 167,A -5.4594,B 11.338,C 0.1328,E1 11.4976,E2 456.0323} C_DIS
LIN {X 130.433,Y -16.4805,Z 167,A -6.8676,B 11.338,C 0.1373,E1 11.4972,E2 457.4436} C_DIS
LIN {X 129.9893,Y -19.6723,Z 167,A -8.249,B 11.3379,C 0.1408,E1 11.4966,E2 458.8239} C_DIS
LIN {X 129.4465,Y -22.9706,Z 167,A -9.6576,B 11.3379,C 0.1438,E1 11.496,E2 460.2282} C_DIS
LIN {X 128.895,Y -25.8877,Z 167,A -11.0059,B 11.3378,C 0.149,E1 11.4952,E2 461.5846} C_DIS
LIN {X 128.1795,Y -29.2235,Z 167,A -12.3213,B 11.3378,C 0.1487,E1 11.4944,E2 462.8811} C_DIS
LIN {X 127.4741,Y -32.1615,Z 167,A -13.763,B 11.3377,C 0.1558,E1 11.4935,E2 464.3392} C_DIS
LIN {X 126.7043,Y -35.0728,Z 167,A -15.0202,B 11.3377,C 0.1582,E1 11.4926,E2 465.5914} C_DIS
LIN {X 125.8082,Y -38.1624,Z 167,A -16.4038,B 11.3376,C 0.1617,E1 11.4915,E2 466.9743} C_DIS
LIN {X 124.8317,Y -41.2442,Z 167,A -17.7946,B 11.3376,C 0.1652,E1 11.4903,E2 468.3646} C_DIS
LIN {X 123.7836,Y -44.2907,Z 167,A -19.1802,B 11.3375,C 0.1687,E1 11.489,E2 469.7495} C_DIS
LIN {X 122.6575,Y -47.3199,Z 167,A -20.5704,B 11.3375,C 0.1721,E1 11.4876,E2 471.1392} C_DIS
LIN {X 121.4606,Y -50.313,Z 167,A -21.957,B 11.3374,C 0.1755,E1 11.4862,E2 472.5253} C_DIS
LIN {X 120.1914,Y -53.2743,Z 167,A -23.3689,B 11.3374,C 0.1796,E1 11.4846,E2 473.9397} C_DIS
LIN {X 118.8205,Y -56.2656,Z 167,A -24.7526,B 11.3373,C 0.1822,E1 11.483,E2 475.319} C_DIS
LIN {X 117.4195,Y -59.1346,Z 167,A -26.2352,B 11.3372,C 0.1883,E1 11.4811,E2 476.8141} C_DIS
LIN {X 115.6885,Y -62.4555,Z 167,A -27.7493,B 11.3372,C 0.1895,E1 11.4791,E2 478.3161} C_DIS
LIN {X 114.3876,Y -64.808,Z 167,A -28.9073,B 11.3372,C 0.1923,E1 11.4776,E2 479.4739} C_DIS
LIN {X 112.764,Y -67.5932,Z 167,A -30.3011,B 11.3371,C 0.1956,E1 11.4756,E2 480.8679} C_DIS
LIN {X 110.8628,Y -70.6679,Z 167,A -31.9729,B 11.3369,C 0.2022,E1 11.4731,E2 482.553} C_DIS
LIN {X 108.4023,Y -74.3866,Z 167,A -33.8413,B 11.3369,C 0.2051,E1 11.4702,E2 484.4147} C_DIS
LIN {X 106.5459,Y -77.0223,Z 167,A -35.1606,B 11.3369,C 0.2063,E1 11.468,E2 485.7252} C_DIS
LIN {X 104.2564,Y -80.0945,Z 167,A -36.8456,B 11.3368,C 0.2108,E1 11.4652,E2 487.414} C_DIS
LIN {X 101.7363,Y -83.2717,Z 167,A -38.6247,B 11.3368,C 0.2152,E1 11.4621,E2 489.1965} C_DIS
LIN {X 99.0142,Y -86.4906,Z 167,A -40.4174,B 11.3367,C 0.2183,E1 11.4588,E2 490.9858} C_DIS
LIN {X 96.3205,Y -89.4808,Z 167,A -42.1585,B 11.3366,C 0.222,E1 11.4556,E2 492.7273} C_DIS
LIN {X 93.512,Y -92.4124,Z 167,A -43.9962,B 11.3365,C 0.2276,E1 11.452,E2 494.5752} C_DIS
LIN {X 90.5013,Y -95.363,Z 167,A -45.8192,B 11.3365,C 0.2312,E1 11.4483,E2 496.3985} C_DIS
LIN {X 87.231,Y -98.3628,Z 167,A -47.6469,B 11.3364,C 0.2324,E1 11.4445,E2 498.2155} C_DIS
LIN {X 84.1575,Y -101.0055,Z 167,A -49.4016,B 11.3364,C 0.2357,E1 11.4408,E2 499.9706} C_DIS
LIN {X 80.8752,Y -103.6523,Z 167,A -51.2697,B 11.3362,C 0.24,E1 11.4367,E2 501.8442} C_DIS
LIN {X 77.4435,Y -106.2406,Z 167,A -53.1496,B 11.3362,C 0.2436,E1 11.4325,E2 503.7267} C_DIS
LIN {X 74.0608,Y -108.626,Z 167,A -54.8935,B 11.3362,C 0.2453,E1 11.4285,E2 505.4653} C_DIS
LIN {X 70.656,Y -110.8703,Z 167,A -56.744,B 11.336,C 0.2502,E1 11.4241,E2 507.3263} C_DIS
LIN {X 67.0014,Y -113.1167,Z 167,A -58.4078,B 11.336,C 0.2481,E1 11.4202,E2 508.9672} C_DIS
LIN {X 64.4614,Y -114.5826,Z 167,A -59.7125,B 11.336,C 0.2508,E1 11.417,E2 510.2762} C_DIS
LIN {X 61.977,Y -115.9456,Z 167,A -61.0357,B 11.336,C 0.2548,E1 11.4137,E2 511.6112} C_DIS
LIN {X 58.77,Y -117.603,Z 167,A -62.4545,B 11.336,C 0.2533,E1 11.4103,E2 513.0128} C_DIS
LIN {X 55.8285,Y -119.0278,Z 167,A -64.06,B 11.3358,C 0.2597,E1 11.4061,E2 514.6414} C_DIS
LIN {X 52.8993,Y -120.3587,Z 167,A -65.3071,B 11.3358,C 0.2577,E1 11.403,E2 515.8711} C_DIS
LIN {X 49.9382,Y -121.6171,Z 167,A -66.7114,B 11.3358,C 0.2596,E1 11.3994,E2 517.2769} C_DIS
LIN {X 47.1587,Y -122.7202,Z 167,A -68.02,B 11.3358,C 0.2612,E1 11.396,E2 518.5871} C_DIS
LIN {X 43.7624,Y -123.9732,Z 167,A -69.5475,B 11.3358,C 0.2618,E1 11.392,E2 520.1099} C_DIS
LIN {X 40.8566,Y -124.9608,Z 167,A -70.9445,B 11.3357,C 0.2647,E1 11.3883,E2 521.5152} C_DIS
LIN {X 37.907,Y -125.8863,Z 167,A -72.2889,B 11.3357,C 0.2659,E1 11.3847,E2 522.8602} C_DIS
LIN {X 33.828,Y -127.0419,Z 167,A -74.1783,B 11.3356,C 0.2686,E1 11.3796,E2 524.7559} C_DIS
LIN {X 30.0238,Y -127.9967,Z 167,A -75.7739,B 11.3356,C 0.2673,E1 11.3753,E2 526.3391} C_DIS
LIN {X 26.8393,Y -128.7014,Z 167,A -77.1401,B 11.3356,C 0.267,E1 11.3716,E2 527.6997} C_DIS
LIN {X 24.0583,Y -129.2501,Z 167,A -78.4264,B 11.3356,C 0.2691,E1 11.368,E2 528.9929} C_DIS
LIN {X 20.8821,Y -129.8019,Z 167,A -79.8726,B 11.3356,C 0.2709,E1 11.364,E2 530.445} C_DIS
LIN {X 17.6782,Y -130.2761,Z 167,A -81.3543,B 11.3355,C 0.2734,E1 11.3599,E2 531.936} C_DIS
LIN {X 14.0952,Y -130.711,Z 167,A -82.723,B 11.3355,C 0.2692,E1 11.3562,E2 533.2811} C_DIS
LIN {X 10.8856,Y -131.0175,Z 167,A -84.1457,B 11.3355,C 0.2702,E1 11.3522,E2 534.7067} C_DIS
LIN {X 8.0601,Y -131.2215,Z 167,A -85.5007,B 11.3355,C 0.2735,E1 11.3484,E2 536.0768} C_DIS
LIN {X 4.825,Y -131.3806,Z 167,A -86.9064,B 11.3355,C 0.2737,E1 11.3444,E2 537.4826} C_DIS
LIN {X 1.6022,Y -131.4604,Z 167,A -88.3625,B 11.3355,C 0.2752,E1 11.3404,E2 538.9455} C_DIS
LIN {X 1.6022,Y -131.4604,Z 167,A -88.3625,B 11.3355,C 0.2752,E1 11.3404,E2 538.9455} C_DIS
Enddeposition()
LIN {X 0.9593,Y -132.3799,Z 167,A -88.2151,B 11.3357,C 0.2719,E1 11.341,E2 538.7814} C_DIS
Startdeposition()
$VEL.CP = VEL_PRINT
LIN {X 3.625,Y -132.3348,Z 167,A -86.7635,B 11.3359,C 0.2645,E1 11.3452,E2 537.293} C_DIS
LIN {X 6.9134,Y -132.204,Z 167,A -85.2036,B 11.3359,C 0.2608,E1 11.3496,E2 535.7158} C_DIS
LIN {X 11.023,Y -131.9247,Z 167,A -83.4647,B 11.3359,C 0.2613,E1 11.3544,E2 533.9812} C_DIS
LIN {X 14.2365,Y -131.6166,Z 167,A -82.1586,B 11.3359,C 0.2629,E1 11.358,E2 532.6855} C_DIS
LIN {X 17.1893,Y -131.2636,Z 167,A -80.7974,B 11.336,C 0.2604,E1 11.3618,E2 531.3144} C_DIS
LIN {X 20.647,Y -130.7648,Z 167,A -79.3507,B 11.336,C 0.2612,E1 11.3658,E2 529.8748} C_DIS
LIN {X 23.6645,Y -130.2524,Z 167,A -78.0208,B 11.336,C 0.2602,E1 11.3695,E2 528.5434} C_DIS
LIN {X 27.53,Y -129.4907,Z 167,A -76.1652,B 11.3361,C 0.2552,E1 11.3746,E2 526.6682} C_DIS
LIN {X 31.4443,Y -128.5963,Z 167,A -74.3811,B 11.3361,C 0.2527,E1 11.3795,E2 524.8772} C_DIS
LIN {X 38.5261,Y -126.6543,Z 167,A -71.3418,B 11.3361,C 0.2532,E1 11.3876,E2 521.8526} C_DIS
LIN {X 43.4725,Y -125.0427,Z 167,A -69.4647,B 11.3361,C 0.2602,E1 11.3925,E2 520.0196} C_DIS
LIN {X 45.5125,Y -124.3163,Z 167,A -68.2653,B 11.3361,C 0.2526,E1 11.3957,E2 518.7874} C_DIS
LIN {X 48.0788,Y -123.3448,Z 167,A -67.0132,B 11.3362,C 0.2496,E1 11.399,E2 517.5263} C_DIS
LIN {X 51.1104,Y -122.1198,Z 167,A -65.6544,B 11.3362,C 0.2492,E1 11.4025,E2 516.1733} C_DIS
LIN {X 54.2767,Y -120.746,Z 167,A -64.1555,B 11.3362,C 0.2471,E1 11.4063,E2 514.6725} C_DIS
LIN {X 57.4474,Y -119.2705,Z 167,A -62.6703,B 11.3363,C 0.2458,E1 11.41,E2 513.1895} C_DIS
LIN {X 60.8054,Y -117.5963,Z 167,A -60.9162,B 11.3364,C 0.2401,E1 11.4144,E2 511.418} C_DIS
LIN {X 64.7911,Y -115.4475,Z 167,A -59.1094,B 11.3364,C 0.241,E1 11.4188,E2 509.6281} C_DIS
LIN {X 67.6321,Y -113.8066,Z 167,A -57.6089,B 11.3365,C 0.2367,E1 11.4225,E2 508.1164} C_DIS
LIN {X 71.1363,Y -111.65,Z 167,A -55.7054,B 11.3366,C 0.2305,E1 11.427,E2 506.1961} C_DIS
LIN {X 74.2756,Y -109.5863,Z 167,A -54.233,B 11.3366,C 0.2317,E1 11.4304,E2 504.741} C_DIS
LIN {X 77.3071,Y -107.4699,Z 167,A -52.6266,B 11.3366,C 0.2286,E1 11.434,E2 503.1323} C_DIS
LIN {X 80.252,Y -105.2885,Z 167,A -51.0384,B 11.3367,C 0.2256,E1 11.4376,E2 501.5422} C_DIS
LIN {X 83.8918,Y -102.4118,Z 167,A -49.1324,B 11.3367,C 0.2243,E1 11.4417,E2 499.6466} C_DIS
LIN {X 86.8699,Y -99.8984,Z 167,A -47.4683,B 11.3368,C 0.2215,E1 11.4452,E2 497.9836} C_DIS
LIN {X 89.9327,Y -97.1507,Z 167,A -45.6017,B 11.3369,C 0.2156,E1 11.4491,E2 496.1045} C_DIS
LIN {X 93.6607,Y -93.5617,Z 167,A -43.4516,B 11.3369,C 0.2131,E1 11.4534,E2 493.963} C_DIS
LIN {X 96.3501,Y -90.7891,Z 167,A -41.7672,B 11.3371,C 0.2091,E1 11.4566,E2 492.2752} C_DIS
LIN {X 99.0855,Y -87.7958,Z 167,A -40.0073,B 11.3371,C 0.205,E1 11.4599,E2 490.5128} C_DIS
LIN {X 102.9424,Y -83.2401,Z 167,A -37.4551,B 11.3372,C 0.1998,E1 11.4645,E2 487.9615} C_DIS
LIN {X 105.8224,Y -79.5468,Z 167,A -35.4971,B 11.3372,C 0.1967,E1 11.4678,E2 486.0098} C_DIS
LIN {X 108.2739,Y -76.176,Z 167,A -33.7516,B 11.3373,C 0.1938,E1 11.4706,E2 484.2693} C_DIS
LIN {X 110.4605,Y -72.9695,Z 167,A -32.026,B 11.3374,C 0.1884,E1 11.4733,E2 482.5362} C_DIS
LIN {X 112.8901,Y -69.151,Z 167,A -30.0863,B 11.3374,C 0.1839,E1 11.4762,E2 480.5966} C_DIS
LIN {X 114.8725,Y -65.8057,Z 167,A -28.1956,B 11.3376,C 0.1739,E1 11.4789,E2 478.6785} C_DIS
LIN {X 116.5044,Y -62.8714,Z 167,A -26.9985,B 11.3376,C 0.177,E1 11.4804,E2 477.5111} C_DIS
LIN {X 120.6609,Y -54.467,Z 167,A -23.2159,B 11.3376,C 0.1734,E1 11.485,E2 473.7577} C_DIS
LIN {X 122.3701,Y -50.5111,Z 167,A -21.1325,B 11.3378,C 0.1624,E1 11.4873,E2 471.6456} C_DIS
LIN {X 124.0406,Y -46.2544,Z 167,A -19.2687,B 11.3378,C 0.16,E1 11.4892,E2 469.7935} C_DIS
LIN {X 125.4293,Y -42.3475,Z 167,A -17.3097,B 11.338,C 0.1505,E1 11.491,E2 467.8124} C_DIS
LIN {X 126.9707,Y -37.4706,Z 167,A -15.2197,B 11.338,C 0.1476,E1 11.4927,E2 465.735} C_DIS
LIN {X 127.9348,Y -34.0329,Z 167,A -13.8016,B 11.338,C 0.1465,E1 11.4937,E2 464.3306} C_DIS
LIN {X 129.3045,Y -28.3922,Z 167,A -11.4519,B 11.338,C 0.1437,E1 11.4952,E2 461.9979} C_DIS
LIN {X 129.9417,Y -25.3168,Z 167,A -9.9322,B 11.3382,C 0.1354,E1 11.4961,E2 460.4572} C_DIS
LIN {X 130.6097,Y -21.6038,Z 167,A -8.2998,B 11.3382,C 0.1306,E1 11.4968,E2 458.8231} C_DIS
LIN {X 131.2199,Y -17.5224,Z 167,A -6.5612,B 11.3382,C 0.1267,E1 11.4975,E2 457.0883} C_DIS
LIN {X 131.6573,Y -13.8579,Z 167,A -5.0786,B 11.3382,C 0.1251,E1 11.498,E2 455.6178} C_DIS
LIN {X 131.938,Y -10.8656,Z 167,A -3.7573,B 11.3383,C 0.1207,E1 11.4983,E2 454.2926} C_DIS
LIN {X 132.1982,Y -7.0297,Z 167,A -2.1098,B 11.3383,C 0.1163,E1 11.4986,E2 452.6453} C_DIS
LIN {X 132.3343,Y -3.6447,Z 167,A -0.6541,B 11.3384,C 0.1122,E1 11.4987,E2 451.1893} C_DIS
LIN {X 132.3861,Y 0.0781,Z 167,A 1.0219,B 11.3384,C 0.1057,E1 11.4987,E2 449.5039} C_DIS
LIN {X 132.3384,Y 3.4954,Z 167,A 2.4719,B 11.3385,C 0.1022,E1 11.4987,E2 448.0558} C_DIS
LIN {X 132.2005,Y 6.9827,Z 167,A 3.8735,B 11.3385,C 0.1006,E1 11.4985,E2 446.6659} C_DIS
LIN {X 132.0273,Y 9.7171,Z 167,A 5.0991,B 11.3385,C 0.0961,E1 11.4982,E2 445.4342} C_DIS
LIN {X 131.6372,Y 14.0448,Z 167,A 6.9282,B 11.3385,C 0.092,E1 11.4977,E2 443.6095} C_DIS
LIN {X 131.22,Y 17.5217,Z 167,A 8.5339,B 11.3386,C 0.0852,E1 11.4972,E2 441.9915} C_DIS
LIN {X 130.583,Y 21.7636,Z 167,A 10.2593,B 11.3386,C 0.0833,E1 11.4964,E2 440.2801} C_DIS
LIN {X 129.9405,Y 25.3232,Z 167,A 11.7541,B 11.3386,C 0.0807,E1 11.4957,E2 438.7924} C_DIS
LIN {X 129.3124,Y 28.3557,Z 167,A 13.2151,B 11.3387,C 0.0736,E1 11.4948,E2 437.3156} C_DIS
LIN {X 128.3223,Y 32.5411,Z 167,A 14.9697,B 11.3387,C 0.0712,E1 11.4936,E2 435.5722} C_DIS
LIN {X 127.1117,Y 36.9892,Z 167,A 17.6201,B 11.3389,C 0.048,E1 11.4915,E2 432.8404} C_DIS
LIN {X 125.5231,Y 42.0659,Z 167,A 19.2358,B 11.3388,C 0.06,E1 11.4902,E2 431.3062} C_DIS
LIN {X 124.3643,Y 45.3793,Z 167,A 20.8231,B 11.3388,C 0.054,E1 11.4887,E2 429.7095} C_DIS
LIN {X 122.8459,Y 49.3398,Z 167,A 22.6165,B 11.3388,C 0.0502,E1 11.4869,E2 427.9197} C_DIS
LIN {X 121.2466,Y 53.1527,Z 167,A 24.2824,B 11.3388,C 0.0487,E1 11.485,E2 426.2673} C_DIS
LIN {X 119.9795,Y 55.9517,Z 167,A 25.6062,B 11.3388,C 0.0453,E1 11.4835,E2 424.9432} C_DIS
LIN {X 118.0026,Y 60.0072,Z 167,A 27.2286,B 11.3388,C 0.0489,E1 11.4816,E2 423.359} C_DIS
LIN {X 116.4881,Y 62.9017,Z 167,A 28.9665,B 11.3388,C 0.0368,E1 11.4792,E2 421.5813} C_DIS
LIN {X 114.5378,Y 66.386,Z 167,A 31.0468,B 11.3389,C 0.0231,E1 11.4763,E2 419.4574} C_DIS
LIN {X 112.5504,Y 69.703,Z 167,A 32.14,B 11.3389,C 0.0343,E1 11.4748,E2 418.433} C_DIS
LIN {X 110.8533,Y 72.3717,Z 167,A 33.7676,B 11.3389,C 0.0242,E1 11.4723,E2 416.7735} C_DIS
LIN {X 108.5834,Y 75.7343,Z 167,A 35.5354,B 11.3389,C 0.0197,E1 11.4695,E2 415.0032} C_DIS
LIN {X 106.2321,Y 78.9985,Z 167,A 37.1844,B 11.3389,C 0.018,E1 11.4667,E2 413.3643} C_DIS
LIN {X 103.6827,Y 82.3161,Z 167,A 39.2558,B 11.3389,C 0.0071,E1 11.4631,E2 411.2606} C_DIS
LIN {X 101.4293,Y 85.0771,Z 167,A 40.3023,B 11.3389,C 0.0166,E1 11.4614,E2 410.2729} C_DIS
LIN {X 99.3386,Y 87.5095,Z 167,A 41.8571,B 11.3389,C 0.0092,E1 11.4585,E2 408.6974} C_DIS
LIN {X 96.5903,Y 90.5346,Z 167,A 43.6425,B 11.3389,C 0.0051,E1 11.4551,E2 406.9093} C_DIS
LIN {X 93.6829,Y 93.5395,Z 167,A 45.4284,B 11.3389,C 0.002,E1 11.4516,E2 405.1255} C_DIS
LIN {X 90.6958,Y 96.4382,Z 167,A 47.2045,B 11.3389,C -0.001,E1 11.448,E2 403.3517} C_DIS
LIN {X 87.6178,Y 99.2429,Z 167,A 48.9968,B 11.3389,C -0.0042,E1 11.4443,E2 401.56} C_DIS
LIN {X 84.1552,Y 102.1961,Z 167,A 51.0464,B 11.3389,C -0.0098,E1 11.4399,E2 399.5002} C_DIS
LIN {X 80.679,Y 104.962,Z 167,A 52.8871,B 11.3389,C -0.0111,E1 11.4358,E2 397.6687} C_DIS
LIN {X 77.3798,Y 107.4175,Z 167,A 54.6708,B 11.3389,C -0.0142,E1 11.4318,E2 395.8842} C_DIS
LIN {X 74.103,Y 109.7032,Z 167,A 56.3981,B 11.3389,C -0.017,E1 11.4278,E2 394.1567} C_DIS
LIN {X 70.6034,Y 111.9874,Z 167,A 58.1448,B 11.3389,C -0.0182,E1 11.4237,E2 392.4171} C_DIS
LIN {X 67.2745,Y 114.0185,Z 167,A 59.8463,B 11.3389,C -0.021,E1 11.4196,E2 390.7138} C_DIS
LIN {X 63.2784,Y 116.2836,Z 167,A 61.8218,B 11.3389,C -0.0234,E1 11.4148,E2 388.7396} C_DIS
LIN {X 59.5012,Y 118.2602,Z 167,A 63.5242,B 11.3389,C -0.0223,E1 11.4106,E2 387.054} C_DIS
LIN {X 56.8791,Y 119.542,Z 167,A 64.7983,B 11.3389,C -0.0241,E1 11.4074,E2 385.7785} C_DIS
LIN {X 53.8969,Y 120.9158,Z 167,A 66.2195,B 11.3389,C -0.0258,E1 11.4038,E2 384.3572} C_DIS
LIN {X 50.2455,Y 122.4807,Z 167,A 68.1044,B 11.3389,C -0.0317,E1 11.3989,E2 382.4528} C_DIS
LIN {X 46.4414,Y 123.9706,Z 167,A 69.6656,B 11.3389,C -0.0284,E1 11.3949,E2 380.9163} C_DIS
LIN {X 43.1881,Y 125.1413,Z 167,A 71.2052,B 11.3389,C -0.0308,E1 11.3908,E2 379.3717} C_DIS
LIN {X 39.534,Y 126.3456,Z 167,A 72.8166,B 11.3389,C -0.0309,E1 11.3866,E2 377.767} C_DIS
LIN {X 36.0429,Y 127.3837,Z 167,A 74.5533,B 11.3389,C -0.036,E1 11.3819,E2 376.0114} C_DIS
LIN {X 32.3431,Y 128.3726,Z 167,A 76.0772,B 11.3389,C -0.034,E1 11.3778,E2 374.5036} C_DIS
LIN {X 29.2568,Y 129.111,Z 167,A 77.3966,B 11.3389,C -0.0335,E1 11.3742,E2 373.1909} C_DIS
LIN {X 26.1041,Y 129.7853,Z 167,A 78.8208,B 11.3389,C -0.0349,E1 11.3703,E2 371.7636} C_DIS
LIN {X 21.9419,Y 130.5533,Z 167,A 80.725,B 11.3389,C -0.0375,E1 11.365,E2 369.8514} C_DIS
LIN {X 17.843,Y 131.1779,Z 167,A 82.5409,B 11.3389,C -0.0387,E1 11.36,E2 368.0336} C_DIS
LIN {X 13.5903,Y 131.6861,Z 167,A 84.2583,B 11.3389,C -0.036,E1 11.3553,E2 366.3329} C_DIS
LIN {X 9.7992,Y 132.0213,Z 167,A 86.0214,B 11.3389,C -0.039,E1 11.3504,E2 364.5567} C_DIS
LIN {X 5.3952,Y 132.2746,Z 167,A 87.8669,B 11.3389,C -0.0377,E1 11.3452,E2 362.7195} C_DIS
LIN {X 1.9569,Y 132.3702,Z 167,A 89.3306,B 11.3389,C -0.0371,E1 11.3412,E2 361.2594} C_DIS
LIN {X -2.3292,Y 132.364,Z 167,A 91.2358,B 11.3389,C -0.0381,E1 11.3358,E2 359.3492} C_DIS
LIN {X -6.6557,Y 132.217,Z 167,A 93.0878,B 11.3389,C -0.0373,E1 11.3307,E2 357.5007} C_DIS
LIN {X -10.8836,Y 131.9365,Z 167,A 94.9765,B 11.3389,C -0.0381,E1 11.3254,E2 355.6065} C_DIS
LIN {X -15.3355,Y 131.4935,Z 167,A 96.8734,B 11.3389,C -0.0365,E1 11.3201,E2 353.7154} C_DIS
LIN {X -19.1833,Y 130.9878,Z 167,A 98.4903,B 11.3389,C -0.0343,E1 11.3157,E2 352.1069} C_DIS
LIN {X -22.9327,Y 130.3834,Z 167,A 100.2119,B 11.3389,C -0.0352,E1 11.3109,E2 350.3771} C_DIS
LIN {X -26.4974,Y 129.7053,Z 167,A 102.1523,B 11.3389,C -0.0426,E1 11.3055,E2 348.394} C_DIS
LIN {X -30.3313,Y 128.8645,Z 167,A 103.3951,B 11.3389,C -0.031,E1 11.3023,E2 347.2064} C_DIS
LIN {X -34.7168,Y 127.7524,Z 167,A 105.4008,B 11.3389,C -0.0305,E1 11.2968,E2 345.1964} C_DIS
LIN {X -38.487,Y 126.6663,Z 167,A 107.5396,B 11.3389,C -0.0389,E1 11.291,E2 343.0067} C_DIS
LIN {X -42.183,Y 125.4841,Z 167,A 108.7346,B 11.3389,C -0.0265,E1 11.288,E2 341.8703} C_DIS
LIN {X -45.4216,Y 124.3491,Z 167,A 110.3225,B 11.3389,C -0.0272,E1 11.2838,E2 340.2716} C_DIS
LIN {X -48.4634,Y 123.1954,Z 167,A 111.6778,B 11.3389,C -0.0244,E1 11.2802,E2 338.9235} C_DIS
LIN {X -51.3099,Y 122.0364,Z 167,A 113.1347,B 11.3389,C -0.0257,E1 11.2765,E2 337.4528} C_DIS
LIN {X -57.5213,Y 119.2352,Z 167,A 116.0367,B 11.3389,C -0.0208,E1 11.2691,E2 334.559} C_DIS
LIN {X -61.2122,Y 117.3827,Z 167,A 118.2033,B 11.3389,C -0.0267,E1 11.2636,E2 332.3491} C_DIS
LIN {X -64.5744,Y 115.5694,Z 167,A 119.9397,B 11.3389,C -0.026,E1 11.2594,E2 330.6043} C_DIS
LIN {X -68.088,Y 113.5349,Z 167,A 121.1869,B 11.3389,C -0.0122,E1 11.2565,E2 329.4192} C_DIS
LIN {X -71.0407,Y 111.7112,Z 167,A 122.8931,B 11.3389,C -0.0142,E1 11.2524,E2 327.6904} C_DIS
LIN {X -74.8236,Y 109.2129,Z 167,A 124.8386,B 11.3389,C -0.0105,E1 11.2479,E2 325.7487} C_DIS
LIN {X -78.4369,Y 106.6474,Z 167,A 126.725,B 11.3389,C -0.0064,E1 11.2437,E2 323.8678} C_DIS
LIN {X -81.8612,Y 104.0421,Z 167,A 128.6513,B 11.3389,C -0.0044,E1 11.2394,E2 321.9359} C_DIS
LIN {X -85.4039,Y 101.1551,Z 167,A 130.6606,B 11.3389,C -0.0012,E1 11.2351,E2 319.9249} C_DIS
LIN {X -88.7193,Y 98.2599,Z 167,A 132.5069,B 11.3389,C 0.0038,E1 11.2313,E2 318.0875} C_DIS
LIN {X -91.5582,Y 95.6197,Z 167,A 134.2655,B 11.3389,C 0.0056,E1 11.2277,E2 316.3211} C_DIS
LIN {X -94.8076,Y 92.3997,Z 167,A 136.2977,B 11.3389,C 0.0087,E1 11.2237,E2 314.2849} C_DIS
LIN {X -97.798,Y 89.2283,Z 167,A 138.1576,B 11.3389,C 0.0134,E1 11.2201,E2 312.4302} C_DIS
LIN {X -100.6069,Y 86.049,Z 167,A 140.0367,B 11.3389,C 0.0167,E1 11.2167,E2 310.5481} C_DIS
LIN {X -103.3853,Y 82.6898,Z 167,A 141.962,B 11.3389,C 0.0203,E1 11.2133,E2 308.6203} C_DIS
LIN {X -106.1412,Y 79.1206,Z 167,A 143.8934,B 11.3389,C 0.0253,E1 11.2101,E2 306.6934} C_DIS
LIN {X -108.4726,Y 75.8936,Z 167,A 145.5424,B 11.3389,C 0.0311,E1 11.2074,E2 305.0551} C_DIS
LIN {X -110.5087,Y 72.8962,Z 167,A 147.5443,B 11.3389,C 0.026,E1 11.2042,E2 303.0035} C_DIS
LIN {X -112.5691,Y 69.673,Z 167,A 148.9166,B 11.3389,C 0.036,E1 11.2023,E2 301.6667} C_DIS
LIN {X -114.604,Y 66.2717,Z 167,A 150.6138,B 11.3389,C 0.0408,E1 11.1999,E2 299.9737} C_DIS
LIN {X -116.3785,Y 63.1044,Z 167,A 152.2215,B 11.3389,C 0.0442,E1 11.1977,E2 298.3634} C_DIS
LIN {X -117.9521,Y 60.1065,Z 167,A 153.686,B 11.3389,C 0.0481,E1 11.1958,E2 296.9006} C_DIS
LIN {X -120.0024,Y 55.9023,Z 167,A 155.4797,B 11.3389,C 0.0582,E1 11.1937,E2 295.1365} C_DIS
LIN {X -122.1972,Y 50.9249,Z 167,A 157.8032,B 11.3388,C 0.0653,E1 11.1911,E2 292.8194} C_DIS
LIN {X -123.2931,Y 48.2119,Z 167,A 159.3428,B 11.3388,C 0.0632,E1 11.1895,E2 291.249} C_DIS
LIN {X -124.5136,Y 44.9655,Z 167,A 160.8925,B 11.3388,C 0.0664,E1 11.188,E2 289.6953} C_DIS
LIN {X -125.8283,Y 41.1494,Z 167,A 162.598,B 11.3388,C 0.0722,E1 11.1865,E2 287.9967} C_DIS
LIN {X -126.5988,Y 38.7076,Z 167,A 163.7207,B 11.3388,C 0.075,E1 11.1855,E2 286.8735} C_DIS
LIN {X -127.6317,Y 35.1563,Z 167,A 165.3642,B 11.3387,C 0.0787,E1 11.1843,E2 285.2268} C_DIS
LIN {X -128.6689,Y 31.1429,Z 167,A 167.6954,B 11.3387,C 0.0729,E1 11.1827,E2 282.8336} C_DIS
LIN {X -129.6254,Y 26.8902,Z 167,A 168.9797,B 11.3386,C 0.0907,E1 11.182,E2 281.6232} C_DIS
LIN {X -130.2571,Y 23.6379,Z 167,A 171.0071,B 11.3386,C 0.0827,E1 11.1809,E2 279.5267} C_DIS
LIN {X -130.9316,Y 19.5698,Z 167,A 172.8802,B 11.3386,C 0.0861,E1 11.1802,E2 277.6451} C_DIS
LIN {X -131.4943,Y 15.329,Z 167,A 174.2175,B 11.3386,C 0.102,E1 11.1797,E2 276.3711} C_DIS
LIN {X -131.8864,Y 11.4766,Z 167,A 175.9692,B 11.3385,C 0.1054,E1 11.1793,E2 274.6123} C_DIS
LIN {X -132.1445,Y 7.9678,Z 167,A 177.5496,B 11.3385,C 0.1087,E1 11.179,E2 273.0266} C_DIS
LIN {X -132.3335,Y 3.6733,Z 167,A 179.3687,B 11.3384,C 0.115,E1 11.1788,E2 271.2144} C_DIS
LIN {X -132.3849,Y -0.3097,Z 167,A -178.821,B 11.3384,C 0.1184,E1 11.1788,E2 269.3957} C_DIS
LIN {X -132.3171,Y -4.2632,Z 167,A -177.0305,B 11.3384,C 0.1218,E1 11.1788,E2 267.5975} C_DIS
LIN {X -132.126,Y -8.2678,Z 167,A -175.3885,B 11.3382,C 0.1288,E1 11.1791,E2 265.9684} C_DIS
LIN {X -131.8083,Y -12.3401,Z 167,A -173.5769,B 11.3382,C 0.133,E1 11.1796,E2 264.1533} C_DIS
LIN {X -131.4366,Y -15.8122,Z 167,A -172.0342,B 11.3382,C 0.1368,E1 11.1801,E2 262.6084} C_DIS
LIN {X -130.8547,Y -20.0663,Z 167,A -169.3848,B 11.3382,C 0.1259,E1 11.1812,E2 259.8656} C_DIS
LIN {X -129.8407,Y -25.8321,Z 167,A -167.7287,B 11.338,C 0.1513,E1 11.182,E2 258.3176} C_DIS
LIN {X -129.215,Y -28.8014,Z 167,A -166.1588,B 11.338,C 0.1498,E1 11.183,E2 256.7182} C_DIS
LIN {X -127.5864,Y -35.318,Z 167,A -163.5418,B 11.3378,C 0.1639,E1 11.1848,E2 254.1385} C_DIS
LIN {X -126.9344,Y -37.5946,Z 167,A -162.3468,B 11.3378,C 0.1633,E1 11.1857,E2 252.9242} C_DIS
LIN {X -125.8913,Y -40.9561,Z 167,A -160.7876,B 11.3378,C 0.1668,E1 11.187,E2 251.3621} C_DIS
LIN {X -125.0218,Y -43.5326,Z 167,A -159.5912,B 11.3378,C 0.1696,E1 11.1881,E2 250.1641} C_DIS
LIN {X -123.906,Y -46.614,Z 167,A -158.1096,B 11.3377,C 0.1722,E1 11.1896,E2 248.6762} C_DIS
LIN {X -122.4755,Y -50.2587,Z 167,A -156.4252,B 11.3376,C 0.177,E1 11.1913,E2 246.9945} C_DIS
LIN {X -120.4766,Y -54.8766,Z 167,A -153.7262,B 11.3376,C 0.1718,E1 11.1945,E2 244.2342} C_DIS
LIN {X -118.7322,Y -58.5504,Z 167,A -152.761,B 11.3373,C 0.193,E1 11.1955,E2 243.366} C_DIS
LIN {X -117.7358,Y -60.5313,Z 167,A -151.4777,B 11.3374,C 0.1887,E1 11.1972,E2 242.0447} C_DIS
LIN {X -116.2017,Y -63.4286,Z 167,A -149.9819,B 11.3374,C 0.1907,E1 11.1992,E2 240.5406} C_DIS
LIN {X -114.1761,Y -67.0062,Z 167,A -148.1371,B 11.3374,C 0.1938,E1 11.2018,E2 238.6891} C_DIS
LIN {X -111.955,Y -70.6547,Z 167,A -146.22,B 11.3373,C 0.1969,E1 11.2046,E2 236.765} C_DIS
LIN {X -109.4756,Y -74.4391,Z 167,A -144.2875,B 11.3372,C 0.2021,E1 11.2076,E2 234.8368} C_DIS
LIN {X -107.3711,Y -77.4438,Z 167,A -142.6806,B 11.3372,C 0.2054,E1 11.2102,E2 233.2285} C_DIS
LIN {X -104.8287,Y -80.8521,Z 167,A -140.8122,B 11.3371,C 0.2089,E1 11.2134,E2 231.3577} C_DIS
LIN {X -101.9491,Y -84.4535,Z 167,A -138.8026,B 11.337,C 0.2131,E1 11.2169,E2 229.3474} C_DIS
LIN {X -98.9438,Y -87.9561,Z 167,A -136.8312,B 11.3369,C 0.2179,E1 11.2205,E2 227.3801} C_DIS
LIN {X -96.0406,Y -91.1172,Z 167,A -134.9148,B 11.3369,C 0.2205,E1 11.2242,E2 225.4575} C_DIS
LIN {X -92.9379,Y -94.2797,Z 167,A -132.9693,B 11.3368,C 0.2237,E1 11.228,E2 223.5094} C_DIS
LIN {X -89.8503,Y -97.2268,Z 167,A -131.1048,B 11.3368,C 0.2269,E1 11.2318,E2 221.6435} C_DIS
LIN {X -86.3224,Y -100.3716,Z 167,A -129.0676,B 11.3366,C 0.2308,E1 11.2361,E2 219.6079} C_DIS
LIN {X -82.8304,Y -103.2728,Z 167,A -127.0416,B 11.3366,C 0.233,E1 11.2405,E2 217.5752} C_DIS
LIN {X -79.4779,Y -105.8744,Z 167,A -125.2892,B 11.3365,C 0.2379,E1 11.2444,E2 215.8335} C_DIS
LIN {X -76.6086,Y -107.9688,Z 167,A -123.6991,B 11.3365,C 0.2392,E1 11.248,E2 214.2373} C_DIS
LIN {X -73.767,Y -109.9298,Z 167,A -122.1316,B 11.3365,C 0.2399,E1 11.2516,E2 212.6612} C_DIS
LIN {X -70.0723,Y -112.3206,Z 167,A -120.2337,B 11.3364,C 0.2429,E1 11.2561,E2 210.7644} C_DIS
LIN {X -66.1013,Y -114.7027,Z 167,A -118.2362,B 11.3364,C 0.2458,E1 11.2609,E2 208.768} C_DIS
LIN {X -62.3805,Y -116.7681,Z 167,A -116.4645,B 11.3362,C 0.2498,E1 11.2652,E2 207.0049} C_DIS
LIN {X -59.2789,Y -118.3727,Z 167,A -114.7807,B 11.3362,C 0.2477,E1 11.2695,E2 205.3002} C_DIS
LIN {X -55.4891,Y -120.1934,Z 167,A -113.1145,B 11.3362,C 0.2532,E1 11.2736,E2 203.6527} C_DIS
LIN {X -52.1089,Y -121.6979,Z 167,A -111.563,B 11.3362,C 0.2561,E1 11.2776,E2 202.1073} C_DIS
LIN {X -49.1583,Y -122.9191,Z 167,A -110.1851,B 11.3361,C 0.2575,E1 11.2811,E2 200.7297} C_DIS
LIN {X -46.2299,Y -124.0498,Z 167,A -108.7288,B 11.3361,C 0.2565,E1 11.285,E2 199.2615} C_DIS
LIN {X -42.3583,Y -125.4257,Z 167,A -107.0888,B 11.336,C 0.2612,E1 11.2893,E2 197.6382} C_DIS
LIN {X -39.3464,Y -126.4033,Z 167,A -105.4131,B 11.3361,C 0.2552,E1 11.2938,E2 195.925} C_DIS
LIN {X -35.3987,Y -127.5639,Z 167,A -103.8278,B 11.336,C 0.261,E1 11.298,E2 194.3633} C_DIS
LIN {X -32.2916,Y -128.3857,Z 167,A -102.3962,B 11.336,C 0.2609,E1 11.3019,E2 192.9265} C_DIS
LIN {X -28.0801,Y -129.3719,Z 167,A -100.5458,B 11.336,C 0.2624,E1 11.3069,E2 191.0783} C_DIS
LIN {X -24.8419,Y -130.0325,Z 167,A -99.0661,B 11.336,C 0.2618,E1 11.311,E2 189.5921} C_DIS
LIN {X -21.6524,Y -130.6016,Z 167,A -97.6991,B 11.336,C 0.2632,E1 11.3148,E2 188.2291} C_DIS
LIN {X -18.4894,Y -131.0869,Z 167,A -96.3389,B 11.336,C 0.2642,E1 11.3185,E2 186.8715} C_DIS
LIN {X -15.4147,Y -131.4841,Z 167,A -95.0307,B 11.3359,C 0.2653,E1 11.3221,E2 185.5669} C_DIS
LIN {X -12.0577,Y -131.8354,Z 167,A -93.3684,B 11.3359,C 0.2607,E1 11.3268,E2 183.8795} C_DIS
LIN {X -7.9681,Y -132.1445,Z 167,A -91.7487,B 11.3359,C 0.2645,E1 11.3313,E2 182.278} C_DIS
LIN {X -4.1152,Y -132.3212,Z 167,A -89.9697,B 11.3359,C 0.2619,E1 11.3363,E2 180.4849} C_DIS
LIN {X 0.1206,Y -132.3858,Z 167,A -88.2528,B 11.3359,C 0.2645,E1 11.341,E2 178.7815} C_DIS
LIN {X 0.1206,Y -132.3858,Z 167,A -88.2528,B 11.3359,C 0.2645,E1 11.341,E2 178.7815} C_DIS
Enddeposition()
LIN {X 0.9608,Y -133.2963,Z 167,A -88.4553,B 11.3349,C 0.2849,E1 11.3397,E2 179.0878} C_DIS
Startdeposition()
$VEL.CP = VEL_PRINT
LIN {X -2.3,Y -133.2802,Z 167,A -89.989,B 11.3349,C 0.2882,E1 11.3354,E2 180.6383} C_DIS
LIN {X -6.3966,Y -133.1467,Z 167,A -91.7374,B 11.3349,C 0.2879,E1 11.3305,E2 182.3858} C_DIS
LIN {X -10.4049,Y -132.8951,Z 167,A -93.4938,B 11.3349,C 0.2885,E1 11.3256,E2 184.1466} C_DIS
LIN {X -13.9604,Y -132.5672,Z 167,A -94.9697,B 11.3349,C 0.2869,E1 11.3215,E2 185.6159} C_DIS
LIN {X -17.4952,Y -132.1469,Z 167,A -96.4854,B 11.3349,C 0.2862,E1 11.3173,E2 187.1304} C_DIS
LIN {X -21.4021,Y -131.5716,Z 167,A -98.2326,B 11.3349,C 0.2868,E1 11.3125,E2 188.8842} C_DIS
LIN {X -25.1333,Y -130.9089,Z 167,A -99.7796,B 11.3349,C 0.2842,E1 11.3083,E2 190.4216} C_DIS
LIN {X -28.7766,Y -130.1582,Z 167,A -101.5231,B 11.3349,C 0.2868,E1 11.3035,E2 192.1832} C_DIS
LIN {X -32.4809,Y -129.2822,Z 167,A -103.0511,B 11.3349,C 0.2834,E1 11.2993,E2 193.6983} C_DIS
LIN {X -36.1939,Y -128.2922,Z 167,A -104.7243,B 11.3349,C 0.2828,E1 11.2948,E2 195.3744} C_DIS
LIN {X -41.5968,Y -126.6443,Z 167,A -107.0055,B 11.3351,C 0.2776,E1 11.2888,E2 197.6382} C_DIS
LIN {X -45.3589,Y -125.345,Z 167,A -108.8515,B 11.3351,C 0.2792,E1 11.2839,E2 199.5007} C_DIS
LIN {X -49.0441,Y -123.9519,Z 167,A -110.6332,B 11.3351,C 0.2797,E1 11.2792,E2 201.2934} C_DIS
LIN {X -52.1487,Y -122.6782,Z 167,A -112.1205,B 11.3351,C 0.2792,E1 11.2754,E2 202.7861} C_DIS
LIN {X -55.3617,Y -121.261,Z 167,A -113.6006,B 11.3351,C 0.2769,E1 11.2716,E2 204.2627} C_DIS
LIN {X -58.8254,Y -119.6174,Z 167,A -115.2511,B 11.3351,C 0.275,E1 11.2675,E2 205.9134} C_DIS
LIN {X -62.0057,Y -118.0001,Z 167,A -116.7288,B 11.3353,C 0.2719,E1 11.2638,E2 207.3842} C_DIS
LIN {X -65.6269,Y -116.0281,Z 167,A -118.5158,B 11.3353,C 0.2699,E1 11.2594,E2 209.173} C_DIS
LIN {X -70.7588,Y -112.9717,Z 167,A -121.1505,B 11.3353,C 0.2678,E1 11.2531,E2 211.8155} C_DIS
LIN {X -74.3794,Y -110.6216,Z 167,A -123.0639,B 11.3353,C 0.2662,E1 11.2487,E2 213.7355} C_DIS
LIN {X -78.1648,Y -107.9794,Z 167,A -125.038,B 11.3355,C 0.2628,E1 11.2442,E2 215.708} C_DIS
LIN {X -81.6769,Y -105.3478,Z 167,A -126.8815,B 11.3355,C 0.2587,E1 11.2401,E2 217.5458} C_DIS
LIN {X -84.9348,Y -102.7393,Z 167,A -129.0821,B 11.3355,C 0.2644,E1 11.2352,E2 219.7947} C_DIS
LIN {X -87.9645,Y -100.1584,Z 167,A -130.5125,B 11.3356,C 0.2552,E1 11.2323,E2 221.191} C_DIS
LIN {X -91.2461,Y -97.1777,Z 167,A -132.4284,B 11.3357,C 0.2518,E1 11.2283,E2 223.1075} C_DIS
LIN {X -94.5412,Y -93.9746,Z 167,A -134.3789,B 11.3358,C 0.2473,E1 11.2245,E2 225.0541} C_DIS
LIN {X -97.6704,Y -90.7182,Z 167,A -136.3275,B 11.3358,C 0.2435,E1 11.2207,E2 227.0028} C_DIS
LIN {X -100.6406,Y -87.4119,Z 167,A -138.2746,B 11.336,C 0.2402,E1 11.2171,E2 228.9535} C_DIS
LIN {X -103.4432,Y -84.0767,Z 167,A -140.1819,B 11.336,C 0.2368,E1 11.2137,E2 230.864} C_DIS
LIN {X -105.5935,Y -81.3598,Z 167,A -141.6944,B 11.336,C 0.234,E1 11.2111,E2 232.3784} C_DIS
LIN {X -108.1905,Y -77.8733,Z 167,A -143.5104,B 11.3362,C 0.2286,E1 11.2082,E2 234.1871} C_DIS
LIN {X -110.438,Y -74.6506,Z 167,A -145.5958,B 11.3362,C 0.2329,E1 11.2048,E2 236.3189} C_DIS
LIN {X -112.5815,Y -71.3775,Z 167,A -146.9543,B 11.3363,C 0.2221,E1 11.2028,E2 237.6377} C_DIS
LIN {X -114.6728,Y -67.9672,Z 167,A -148.7071,B 11.3364,C 0.2185,E1 11.2003,E2 239.3934} C_DIS
LIN {X -116.8234,Y -64.2005,Z 167,A -150.5832,B 11.3364,C 0.2141,E1 11.1977,E2 241.2697} C_DIS
LIN {X -118.5947,Y -60.8623,Z 167,A -152.1096,B 11.3366,C 0.2079,E1 11.1958,E2 242.7831} C_DIS
LIN {X -120.5802,Y -56.8289,Z 167,A -154.2859,B 11.3366,C 0.2079,E1 11.1931,E2 244.9872} C_DIS
LIN {X -122.3234,Y -52.9691,Z 167,A -155.921,B 11.3368,C 0.1993,E1 11.1913,E2 246.5986} C_DIS
LIN {X -123.6109,Y -49.8909,Z 167,A -157.4348,B 11.3368,C 0.1971,E1 11.1897,E2 248.1208} C_DIS
LIN {X -125.1042,Y -46.025,Z 167,A -159.3388,B 11.3368,C 0.1948,E1 11.1878,E2 250.0382} C_DIS
LIN {X -126.3224,Y -42.5635,Z 167,A -160.8543,B 11.3369,C 0.1892,E1 11.1864,E2 251.5449} C_DIS
LIN {X -127.3609,Y -39.3458,Z 167,A -162.3937,B 11.3369,C 0.1869,E1 11.1851,E2 253.0933} C_DIS
LIN {X -128.4662,Y -35.5715,Z 167,A -164.6948,B 11.3369,C 0.1946,E1 11.1834,E2 255.4652} C_DIS
LIN {X -129.8133,Y -30.2926,Z 167,A -166.3954,B 11.3371,C 0.1749,E1 11.1823,E2 257.0879} C_DIS
LIN {X -130.9865,Y -24.727,Z 167,A -169.2539,B 11.3371,C 0.1763,E1 11.1807,E2 259.9931} C_DIS
LIN {X -131.662,Y -20.8363,Z 167,A -170.6131,B 11.3373,C 0.1646,E1 11.1801,E2 261.3106} C_DIS
LIN {X -132.2131,Y -16.9896,Z 167,A -172.3639,B 11.3373,C 0.1613,E1 11.1794,E2 263.0693} C_DIS
LIN {X -132.6542,Y -13.1091,Z 167,A -174.0236,B 11.3374,C 0.1561,E1 11.1789,E2 264.7251} C_DIS
LIN {X -133.0136,Y -8.7499,Z 167,A -175.9136,B 11.3374,C 0.1508,E1 11.1786,E2 266.6144} C_DIS
LIN {X -133.204,Y -5.0584,Z 167,A -177.4611,B 11.3376,C 0.1453,E1 11.1784,E2 268.1554} C_DIS
LIN {X -133.2969,Y -0.9661,Z 167,A -179.2587,B 11.3376,C 0.1409,E1 11.1783,E2 269.9557} C_DIS
LIN {X -133.2684,Y 2.9873,Z 167,A 178.963,B 11.3376,C 0.1375,E1 11.1783,E2 271.7417} C_DIS
LIN {X -133.1543,Y 6.2462,Z 167,A 177.6659,B 11.3377,C 0.1312,E1 11.1785,E2 273.0248} C_DIS
LIN {X -132.952,Y 9.6247,Z 167,A 176.152,B 11.3377,C 0.1281,E1 11.1788,E2 274.5441} C_DIS
LIN {X -132.6271,Y 13.3917,Z 167,A 174.4588,B 11.3378,C 0.1248,E1 11.1792,E2 276.2437} C_DIS
LIN {X -132.1882,Y 17.1801,Z 167,A 172.9664,B 11.3378,C 0.117,E1 11.1797,E2 277.7168} C_DIS
LIN {X -131.6472,Y 20.9318,Z 167,A 170.5781,B 11.3378,C 0.1275,E1 11.1808,E2 280.1928} C_DIS
LIN {X -130.798,Y 25.7137,Z 167,A 168.9613,B 11.3379,C 0.112,E1 11.1816,E2 281.752} C_DIS
LIN {X -129.6876,Y 30.8237,Z 167,A 166.606,B 11.3379,C 0.1077,E1 11.183,E2 284.1174} C_DIS
LIN {X -128.4379,Y 35.6727,Z 167,A 164.5971,B 11.3381,C 0.0986,E1 11.1845,E2 286.107} C_DIS
LIN {X -127.5034,Y 38.8802,Z 167,A 163.1361,B 11.3381,C 0.095,E1 11.1856,E2 287.5692} C_DIS
LIN {X -126.4284,Y 42.2451,Z 167,A 161.6153,B 11.3381,C 0.0908,E1 11.187,E2 289.0887} C_DIS
LIN {X -125.1524,Y 45.893,Z 167,A 159.7989,B 11.3381,C 0.0893,E1 11.1887,E2 290.9215} C_DIS
LIN {X -123.7093,Y 49.6467,Z 167,A 158.1794,B 11.3381,C 0.0823,E1 11.1903,E2 292.5261} C_DIS
LIN {X -121.9983,Y 53.7187,Z 167,A 156.0302,B 11.3381,C 0.0823,E1 11.1927,E2 294.7028} C_DIS
LIN {X -120.1657,Y 57.6976,Z 167,A 154.2717,B 11.3382,C 0.0746,E1 11.1948,E2 296.4443} C_DIS
LIN {X -118.1789,Y 61.6651,Z 167,A 152.4405,B 11.3382,C 0.068,E1 11.1971,E2 298.2645} C_DIS
LIN {X -116.1987,Y 65.3234,Z 167,A 150.5874,B 11.3382,C 0.0647,E1 11.1996,E2 300.1233} C_DIS
LIN {X -114.3091,Y 68.5772,Z 167,A 148.2806,B 11.3382,C 0.0746,E1 11.203,E2 302.5089} C_DIS
LIN {X -111.5012,Y 73.0537,Z 167,A 146.5867,B 11.3383,C 0.0571,E1 11.2055,E2 304.1329} C_DIS
LIN {X -109.0758,Y 76.6277,Z 167,A 144.7478,B 11.3383,C 0.0522,E1 11.2084,E2 305.9675} C_DIS
LIN {X -106.6857,Y 79.9224,Z 167,A 142.9109,B 11.3383,C 0.0498,E1 11.2115,E2 307.8127} C_DIS
LIN {X -103.9674,Y 83.4276,Z 167,A 141.0193,B 11.3383,C 0.045,E1 11.2147,E2 309.7004} C_DIS
LIN {X -101.3172,Y 86.627,Z 167,A 139.1842,B 11.3384,C 0.0419,E1 11.218,E2 311.5395} C_DIS
LIN {X -98.3448,Y 89.987,Z 167,A 137.2339,B 11.3384,C 0.0381,E1 11.2217,E2 313.4903} C_DIS
LIN {X -95.3434,Y 93.1609,Z 167,A 135.3719,B 11.3384,C 0.0337,E1 11.2253,E2 315.3483} C_DIS
LIN {X -92.3091,Y 96.1685,Z 167,A 133.4937,B 11.3384,C 0.0307,E1 11.229,E2 317.2295} C_DIS
LIN {X -89.0594,Y 99.1853,Z 167,A 131.5748,B 11.3384,C 0.0271,E1 11.233,E2 319.1479} C_DIS
LIN {X -85.698,Y 102.1035,Z 167,A 129.6836,B 11.3384,C 0.0229,E1 11.237,E2 321.0346} C_DIS
LIN {X -82.29,Y 104.8695,Z 167,A 127.7503,B 11.3384,C 0.0204,E1 11.2412,E2 322.9714} C_DIS
LIN {X -78.6761,Y 107.6078,Z 167,A 125.7652,B 11.3384,C 0.0176,E1 11.2457,E2 324.9588} C_DIS
LIN {X -75.1549,Y 110.0959,Z 167,A 123.9197,B 11.3384,C 0.0142,E1 11.2499,E2 326.8016} C_DIS
LIN {X -71.6179,Y 112.4288,Z 167,A 122.0826,B 11.3384,C 0.0116,E1 11.2542,E2 328.6388} C_DIS
LIN {X -67.8711,Y 114.7299,Z 167,A 120.2108,B 11.3384,C 0.0082,E1 11.2587,E2 330.5068} C_DIS
LIN {X -63.7119,Y 117.09,Z 167,A 117.6365,B 11.3384,C 0.0163,E1 11.2651,E2 333.1397} C_DIS
LIN {X -59.6011,Y 119.2348,Z 167,A 116.0882,B 11.3384,C 0.004,E1 11.2688,E2 334.6344} C_DIS
LIN {X -55.0906,Y 121.3843,Z 167,A 113.8061,B 11.3384,C 0.0042,E1 11.2746,E2 336.9304} C_DIS
LIN {X -50.2332,Y 123.4729,Z 167,A 111.7036,B 11.3384,C -0.0023,E1 11.28,E2 339.0111} C_DIS
LIN {X -46.7209,Y 124.8436,Z 167,A 110.1903,B 11.3384,C -0.0064,E1 11.2839,E2 340.5105} C_DIS
LIN {X -42.7482,Y 126.2609,Z 167,A 108.3758,B 11.3384,C -0.0082,E1 11.2887,E2 342.3238} C_DIS
LIN {X -34.9731,Y 128.6316,Z 167,A 104.8476,B 11.3384,C -0.0105,E1 11.2982,E2 345.8536} C_DIS
LIN {X -26.6417,Y 130.6103,Z 167,A 101.1155,B 11.3384,C -0.012,E1 11.3083,E2 349.5892} C_DIS
LIN {X -23.4717,Y 131.217,Z 167,A 99.7492,B 11.3384,C -0.0133,E1 11.312,E2 350.9523} C_DIS
LIN {X -20.1171,Y 131.7733,Z 167,A 98.2052,B 11.3384,C -0.0122,E1 11.3163,E2 352.505} C_DIS
LIN {X -15.7813,Y 132.3624,Z 167,A 96.417,B 11.3384,C -0.0151,E1 11.3212,E2 354.2812} C_DIS
LIN {X -12.6207,Y 132.7011,Z 167,A 94.9968,B 11.3384,C -0.0144,E1 11.3252,E2 355.707} C_DIS
LIN {X -8.7058,Y 133.0163,Z 167,A 93.2503,B 11.3384,C -0.0135,E1 11.3301,E2 357.4595} C_DIS
LIN {X -4.7494,Y 133.2161,Z 167,A 91.4816,B 11.3384,C -0.0123,E1 11.335,E2 359.235} C_DIS
LIN {X -0.7681,Y 133.2978,Z 167,A 89.8692,B 11.3384,C -0.0147,E1 11.3395,E2 360.8349} C_DIS
LIN {X 3.171,Y 133.2633,Z 167,A 88.079,B 11.3384,C -0.0125,E1 11.3445,E2 362.6359} C_DIS
LIN {X 7.2338,Y 133.1046,Z 167,A 86.3453,B 11.3384,C -0.0126,E1 11.3494,E2 364.3672} C_DIS
LIN {X 11.1071,Y 132.8364,Z 167,A 84.7618,B 11.3384,C -0.0143,E1 11.3537,E2 365.94} C_DIS
LIN {X 15.0692,Y 132.4473,Z 167,A 82.9405,B 11.3384,C -0.0113,E1 11.3588,E2 367.7737} C_DIS
LIN {X 18.9762,Y 131.9422,Z 167,A 81.3614,B 11.3384,C -0.0134,E1 11.3632,E2 369.3387} C_DIS
Enddeposition()
END
